KUKA KRL program: MyProgram_263().src

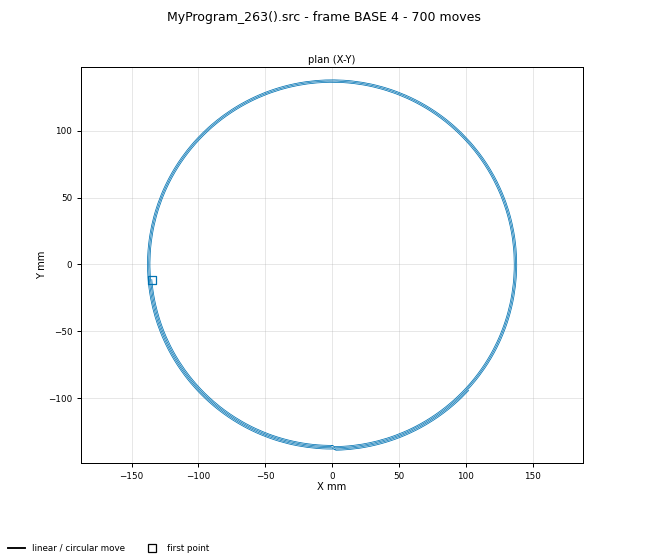
[picture p0: tool path of MyProgram_263().src in frame BASE 4, 700 of 700 moves have a stored position in this frame; points joined in program order, loops and branches not executed]
&ACCESS RVP
&REL 1
&PARAM TEMPLATE = C:\KRC\Roboter\Template\vorgabe
&PARAM EDITMASK = *
DEF MyProgram_263()
; ---- Setting reference (Base) ----
$BASE = BASE_DATA[4]

; --------------------------
; ---- Setting tool (TCP) ----
$TOOL = TOOL_DATA[3]
; --------------------------

$VEL.CP = VEL_APROX_PRINT
Startdeposition()
$VEL.CP = VEL_PRINT
LIN {X -134.8458,Y -11.2904,Z 168,A -173.803,B 10.3704,C 0.1903,E1 10.2126,E2 264.7612} C_DIS
LIN {X -134.4588,Y -15.2399,Z 168,A -171.9605,B 10.3704,C 0.1921,E1 10.2132,E2 262.9003} C_DIS
LIN {X -133.9529,Y -19.1689,Z 168,A -170.374,B 10.3703,C 0.1986,E1 10.2138,E2 261.3266} C_DIS
LIN {X -133.392,Y -22.7512,Z 168,A -168.8018,B 10.3703,C 0.2023,E1 10.2145,E2 259.7513} C_DIS
LIN {X -132.6804,Y -26.5871,Z 168,A -167.1161,B 10.3701,C 0.2064,E1 10.2154,E2 258.0628} C_DIS
LIN {X -131.9635,Y -29.9407,Z 168,A -165.7968,B 10.3701,C 0.213,E1 10.2162,E2 256.7611} C_DIS
LIN {X -130.6956,Y -35.0639,Z 168,A -163.3968,B 10.3699,C 0.2162,E1 10.2178,E2 254.3427} C_DIS
LIN {X -129.3305,Y -39.8048,Z 168,A -161.2288,B 10.3699,C 0.2205,E1 10.2196,E2 252.1668} C_DIS
LIN {X -127.9504,Y -44.0403,Z 168,A -159.3976,B 10.3697,C 0.2267,E1 10.2212,E2 250.3438} C_DIS
LIN {X -126.827,Y -47.1777,Z 168,A -157.8777,B 10.3697,C 0.2284,E1 10.2226,E2 248.8116} C_DIS
LIN {X -125.4357,Y -50.7607,Z 168,A -156.287,B 10.3696,C 0.2335,E1 10.2243,E2 247.2266} C_DIS
LIN {X -123.8895,Y -54.4311,Z 168,A -154.6014,B 10.3695,C 0.238,E1 10.2261,E2 245.5425} C_DIS
LIN {X -120.8002,Y -60.9773,Z 168,A -151.5048,B 10.3693,C 0.2453,E1 10.2299,E2 242.4441} C_DIS
LIN {X -118.8985,Y -64.61,Z 168,A -149.6278,B 10.3693,C 0.247,E1 10.2324,E2 240.551} C_DIS
LIN {X -116.7353,Y -68.4408,Z 168,A -147.7469,B 10.3692,C 0.2512,E1 10.235,E2 238.6689} C_DIS
LIN {X -114.2872,Y -72.4552,Z 168,A -146.0083,B 10.3689,C 0.261,E1 10.2375,E2 236.9629} C_DIS
LIN {X -109.9875,Y -78.8291,Z 168,A -142.3087,B 10.3689,C 0.26,E1 10.2434,E2 233.2102} C_DIS
LIN {X -106.8364,Y -83.0498,Z 168,A -140.2258,B 10.3688,C 0.2679,E1 10.2469,E2 231.1468} C_DIS
LIN {X -104.0676,Y -86.4942,Z 168,A -138.2956,B 10.3687,C 0.2709,E1 10.2503,E2 229.2102} C_DIS
LIN {X -101.2009,Y -89.8315,Z 168,A -136.4119,B 10.3686,C 0.2744,E1 10.2538,E2 227.3247} C_DIS
LIN {X -98.1852,Y -93.1184,Z 168,A -134.4868,B 10.3686,C 0.2776,E1 10.2575,E2 225.3958} C_DIS
LIN {X -95.0955,Y -96.2718,Z 168,A -132.6344,B 10.3684,C 0.2816,E1 10.2611,E2 223.5463} C_DIS
LIN {X -91.911,Y -99.3166,Z 168,A -130.7339,B 10.3684,C 0.2845,E1 10.265,E2 221.642} C_DIS
LIN {X -88.3478,Y -102.4983,Z 168,A -127.9328,B 10.3686,C 0.2721,E1 10.2711,E2 218.7437} C_DIS
LIN {X -83.5517,Y -106.4442,Z 168,A -126.3106,B 10.368,C 0.2976,E1 10.2744,E2 217.2487} C_DIS
LIN {X -80.2823,Y -108.9314,Z 168,A -124.2688,B 10.368,C 0.2942,E1 10.279,E2 215.1697} C_DIS
LIN {X -76.5904,Y -111.5579,Z 168,A -122.3677,B 10.368,C 0.2976,E1 10.2833,E2 213.271} C_DIS
LIN {X -72.4048,Y -114.3191,Z 168,A -119.5332,B 10.3683,C 0.2858,E1 10.2902,E2 210.3474} C_DIS
LIN {X -67.4204,Y -117.3283,Z 168,A -117.9883,B 10.3676,C 0.3086,E1 10.2937,E2 208.9185} C_DIS
LIN {X -64.2373,Y -119.1003,Z 168,A -116.1108,B 10.3678,C 0.3036,E1 10.2984,E2 206.9992} C_DIS
LIN {X -60.1371,Y -121.2202,Z 168,A -114.2859,B 10.3676,C 0.3087,E1 10.3029,E2 205.1905} C_DIS
LIN {X -56.9432,Y -122.7526,Z 168,A -112.8278,B 10.3676,C 0.3112,E1 10.3065,E2 203.7377} C_DIS
LIN {X -51.2127,Y -125.2535,Z 168,A -110.0453,B 10.3676,C 0.3112,E1 10.3137,E2 200.9383} C_DIS
LIN {X -47.9106,Y -126.5525,Z 168,A -108.6757,B 10.3674,C 0.3154,E1 10.3173,E2 199.5851} C_DIS
LIN {X -44.7471,Y -127.7053,Z 168,A -107.1029,B 10.3674,C 0.3134,E1 10.3214,E2 197.9938} C_DIS
LIN {X -40.4758,Y -129.124,Z 168,A -105.146,B 10.3674,C 0.3138,E1 10.3267,E2 196.0302} C_DIS
LIN {X -36.863,Y -130.2001,Z 168,A -103.6169,B 10.3674,C 0.3164,E1 10.3308,E2 194.5092} C_DIS
LIN {X -33.2529,Y -131.1679,Z 168,A -102.06,B 10.3674,C 0.3179,E1 10.3349,E2 192.9552} C_DIS
LIN {X -29.1522,Y -132.1412,Z 168,A -100.2394,B 10.3674,C 0.3181,E1 10.3399,E2 191.1297} C_DIS
LIN {X -25.4818,Y -132.8965,Z 168,A -98.7005,B 10.3673,C 0.3198,E1 10.3441,E2 189.5963} C_DIS
LIN {X -21.682,Y -133.5704,Z 168,A -96.9644,B 10.3673,C 0.3182,E1 10.3489,E2 187.8469} C_DIS
LIN {X -17.6427,Y -134.1624,Z 168,A -95.3562,B 10.3673,C 0.3213,E1 10.3533,E2 186.2533} C_DIS
LIN {X -14.2701,Y -134.5631,Z 168,A -93.9184,B 10.3673,C 0.3216,E1 10.3573,E2 184.8149} C_DIS
LIN {X -10.5281,Y -134.9091,Z 168,A -92.1828,B 10.3673,C 0.3186,E1 10.3622,E2 183.0606} C_DIS
LIN {X -6.8196,Y -135.1457,Z 168,A -90.7307,B 10.3673,C 0.3213,E1 10.3662,E2 181.6231} C_DIS
LIN {X -2.7689,Y -135.2903,Z 168,A -88.9419,B 10.3673,C 0.3196,E1 10.3712,E2 179.8245} C_DIS
LIN {X 0.9792,Y -135.3136,Z 168,A -88.0702,B 10.3668,C 0.3356,E1 10.3735,E2 179.0416} C_DIS
Enddeposition()
LIN {X 0.9792,Y -135.3136,Z 168,A -88.0702,B 10.3668,C 0.3356,E1 10.3735,E2 179.0416} C_DIS
Startdeposition()
$VEL.CP = VEL_PRINT
LIN {X -1.5086,Y -136.2254,Z 168,A -89.0405,B 10.307,C 0.3424,E1 10.311,E2 180.0553} C_DIS
LIN {X -5.484,Y -136.1213,Z 168,A -90.778,B 10.307,C 0.3439,E1 10.3061,E2 181.8016} C_DIS
LIN {X -8.5527,Y -135.963,Z 168,A -92.0736,B 10.307,C 0.3439,E1 10.3025,E2 183.0982} C_DIS
LIN {X -13.1963,Y -135.591,Z 168,A -94.0386,B 10.307,C 0.3438,E1 10.297,E2 185.0647} C_DIS
LIN {X -17.8817,Y -135.0529,Z 168,A -95.9859,B 10.307,C 0.3425,E1 10.2917,E2 187.0081} C_DIS
LIN {X -21.6319,Y -134.5054,Z 168,A -97.5637,B 10.307,C 0.3417,E1 10.2873,E2 188.5845} C_DIS
LIN {X -25.7616,Y -133.7736,Z 168,A -99.3345,B 10.307,C 0.3411,E1 10.2824,E2 190.3565} C_DIS
LIN {X -29.123,Y -133.0826,Z 168,A -100.768,B 10.307,C 0.3402,E1 10.2785,E2 191.7892} C_DIS
LIN {X -32.3071,Y -132.3457,Z 168,A -102.1967,B 10.307,C 0.3406,E1 10.2746,E2 193.225} C_DIS
LIN {X -35.8968,Y -131.4194,Z 168,A -103.7296,B 10.307,C 0.3391,E1 10.2705,E2 194.7551} C_DIS
LIN {X -39.0103,Y -130.5287,Z 168,A -105.0997,B 10.307,C 0.3383,E1 10.2668,E2 196.1263} C_DIS
LIN {X -42.2484,Y -129.5172,Z 168,A -106.5325,B 10.3071,C 0.3374,E1 10.263,E2 197.5601} C_DIS
LIN {X -45.4156,Y -128.4409,Z 168,A -107.9472,B 10.3071,C 0.3364,E1 10.2593,E2 198.976} C_DIS
LIN {X -48.573,Y -127.2804,Z 168,A -109.3701,B 10.3071,C 0.3352,E1 10.2555,E2 200.4} C_DIS
LIN {X -51.7172,Y -126.0356,Z 168,A -110.8009,B 10.3072,C 0.334,E1 10.2518,E2 201.832} C_DIS
LIN {X -54.8451,Y -124.7063,Z 168,A -112.2392,B 10.3072,C 0.3327,E1 10.2481,E2 203.2715} C_DIS
LIN {X -57.4972,Y -123.5035,Z 168,A -113.4678,B 10.3073,C 0.3314,E1 10.245,E2 204.5005} C_DIS
LIN {X -60.8012,Y -121.9117,Z 168,A -115.0386,B 10.3073,C 0.3302,E1 10.2411,E2 206.0748} C_DIS
LIN {X -64.8576,Y -119.8045,Z 168,A -117.0288,B 10.3073,C 0.3292,E1 10.2361,E2 208.0734} C_DIS
LIN {X -68.6292,Y -117.6847,Z 168,A -118.91,B 10.3074,C 0.3281,E1 10.2316,E2 209.9621} C_DIS
LIN {X -72.3466,Y -115.4366,Z 168,A -120.7015,B 10.3075,C 0.3247,E1 10.2273,E2 211.749} C_DIS
LIN {X -75.9181,Y -113.1194,Z 168,A -122.533,B 10.3075,C 0.3229,E1 10.223,E2 213.5853} C_DIS
LIN {X -79.5937,Y -110.5644,Z 168,A -124.4566,B 10.3076,C 0.3207,E1 10.2186,E2 215.5136} C_DIS
LIN {X -83.0341,Y -108.0042,Z 168,A -126.2509,B 10.3077,C 0.3175,E1 10.2146,E2 217.3063} C_DIS
LIN {X -86.5489,Y -105.209,Z 168,A -128.1457,B 10.3078,C 0.3143,E1 10.2105,E2 219.2015} C_DIS
LIN {X -89.9021,Y -102.3584,Z 168,A -130.0271,B 10.3079,C 0.3116,E1 10.2065,E2 221.086} C_DIS
LIN {X -93.1649,Y -99.3979,Z 168,A -131.8853,B 10.308,C 0.3081,E1 10.2027,E2 222.9442} C_DIS
LIN {X -96.3318,Y -96.3318,Z 168,A -133.7845,B 10.3081,C 0.3054,E1 10.1989,E2 224.8484} C_DIS
LIN {X -99.3979,Y -93.1649,Z 168,A -135.6301,B 10.3082,C 0.3015,E1 10.1954,E2 226.6922} C_DIS
LIN {X -102.3584,Y -89.9021,Z 168,A -137.5391,B 10.3082,C 0.2987,E1 10.1918,E2 228.6074} C_DIS
LIN {X -105.209,Y -86.5489,Z 168,A -139.4098,B 10.3084,C 0.295,E1 10.1885,E2 230.4796} C_DIS
LIN {X -107.9455,Y -83.1108,Z 168,A -141.2413,B 10.3085,C 0.2906,E1 10.1853,E2 232.3082} C_DIS
LIN {X -110.5644,Y -79.5937,Z 168,A -143.1423,B 10.3086,C 0.2875,E1 10.1822,E2 234.2152} C_DIS
LIN {X -113.0624,Y -76.0036,Z 168,A -145.0023,B 10.3087,C 0.2835,E1 10.1792,E2 236.0767} C_DIS
LIN {X -115.3278,Y -72.519,Z 168,A -146.7386,B 10.3088,C 0.2791,E1 10.1766,E2 237.8106} C_DIS
LIN {X -117.6847,Y -68.6292,Z 168,A -148.6686,B 10.309,C 0.2747,E1 10.1739,E2 239.7415} C_DIS
LIN {X -119.8045,Y -64.8576,Z 168,A -150.5546,B 10.309,C 0.2715,E1 10.1713,E2 241.6345} C_DIS
LIN {X -121.5696,Y -61.4807,Z 168,A -152.0939,B 10.3092,C 0.2661,E1 10.1694,E2 243.1649} C_DIS
LIN {X -123.2926,Y -57.9533,Z 168,A -153.7231,B 10.3092,C 0.2614,E1 10.1674,E2 244.7903} C_DIS
LIN {X -124.7063,Y -54.8451,Z 168,A -155.1768,B 10.3094,C 0.258,E1 10.1657,E2 246.2451} C_DIS
LIN {X -125.8387,Y -52.1888,Z 168,A -156.4508,B 10.3094,C 0.2559,E1 10.1644,E2 247.5255} C_DIS
LIN {X -127.2804,Y -48.573,Z 168,A -158.0638,B 10.3096,C 0.2511,E1 10.1627,E2 249.1343} C_DIS
LIN {X -128.4409,Y -45.4156,Z 168,A -159.496,B 10.3096,C 0.2476,E1 10.1614,E2 250.5676} C_DIS
LIN {X -129.3486,Y -42.7549,Z 168,A -160.7421,B 10.3096,C 0.2455,E1 10.1602,E2 251.8205} C_DIS
LIN {X -130.5099,Y -39.0744,Z 168,A -162.3371,B 10.3098,C 0.2405,E1 10.1589,E2 253.4107} C_DIS
LIN {X -131.2891,Y -36.3625,Z 168,A -163.5799,B 10.3098,C 0.2382,E1 10.158,E2 254.6594} C_DIS
LIN {X -132.2465,Y -32.7185,Z 168,A -165.1434,B 10.31,C 0.2334,E1 10.1569,E2 256.219} C_DIS
LIN {X -132.8521,Y -30.155,Z 168,A -166.2801,B 10.31,C 0.2308,E1 10.1562,E2 257.3582} C_DIS
LIN {X -133.6569,Y -26.372,Z 168,A -167.9128,B 10.3101,C 0.2263,E1 10.1553,E2 258.9903} C_DIS
LIN {X -134.2422,Y -23.2094,Z 168,A -169.2825,B 10.3101,C 0.2228,E1 10.1546,E2 260.3609} C_DIS
LIN {X -134.9314,Y -18.7824,Z 168,A -171.183,B 10.3103,C 0.2176,E1 10.1538,E2 262.2616} C_DIS
LIN {X -135.2978,Y -15.9235,Z 168,A -172.4765,B 10.3103,C 0.2157,E1 10.1534,E2 263.5639} C_DIS
LIN {X -135.7291,Y -11.6921,Z 168,A -174.2763,B 10.3104,C 0.2107,E1 10.1529,E2 265.3634} C_DIS
LIN {X -135.9751,Y -8.3552,Z 168,A -175.6814,B 10.3105,C 0.2065,E1 10.1526,E2 266.7668} C_DIS
LIN {X -136.1579,Y -4.5455,Z 168,A -177.2807,B 10.3106,C 0.2018,E1 10.1524,E2 268.364} C_DIS
LIN {X -136.2254,Y -1.5086,Z 168,A -178.5008,B 10.3107,C 0.197,E1 10.1524,E2 269.5758} C_DIS
LIN {X -136.2254,Y 1.5086,Z 168,A 179.976,B 10.3107,C 0.198,E1 10.1524,E2 271.1288} C_DIS
LIN {X -136.1281,Y 5.3099,Z 168,A 178.467,B 10.3108,C 0.1917,E1 10.1525,E2 272.6252} C_DIS
LIN {X -135.963,Y 8.5527,Z 168,A 177.0578,B 10.3108,C 0.1885,E1 10.1528,E2 274.0382} C_DIS
LIN {X -135.6827,Y 12.2412,Z 168,A 175.5398,B 10.311,C 0.1832,E1 10.1531,E2 275.5501} C_DIS
LIN {X -135.1791,Y 16.9188,Z 168,A 173.5284,B 10.311,C 0.1781,E1 10.1538,E2 277.5634} C_DIS
LIN {X -134.7492,Y 20.0574,Z 168,A 172.1744,B 10.3111,C 0.1746,E1 10.1543,E2 278.9187} C_DIS
LIN {X -134.2842,Y 22.9573,Z 168,A 170.9468,B 10.3111,C 0.1709,E1 10.1548,E2 280.144} C_DIS
LIN {X -133.7736,Y 25.7616,Z 168,A 169.6915,B 10.3112,C 0.1685,E1 10.1555,E2 281.4049} C_DIS
LIN {X -133.0265,Y 29.383,Z 168,A 168.1143,B 10.3112,C 0.1644,E1 10.1564,E2 282.9831} C_DIS
LIN {X -132.2465,Y 32.7185,Z 168,A 166.6563,B 10.3113,C 0.1607,E1 10.1574,E2 284.4417} C_DIS
LIN {X -131.4194,Y 35.8968,Z 168,A 165.2535,B 10.3113,C 0.1571,E1 10.1584,E2 285.8456} C_DIS
LIN {X -130.5999,Y 38.7669,Z 168,A 163.9581,B 10.3114,C 0.1543,E1 10.1594,E2 287.1446} C_DIS
LIN {X -129.5172,Y 42.2484,Z 168,A 162.4211,B 10.3114,C 0.1501,E1 10.1607,E2 288.6803} C_DIS
LIN {X -128.4409,Y 45.4156,Z 168,A 160.9926,B 10.3115,C 0.1466,E1 10.162,E2 290.11} C_DIS
LIN {X -127.2804,Y 48.573,Z 168,A 159.5563,B 10.3115,C 0.1431,E1 10.1634,E2 291.5473} C_DIS
LIN {X -126.231,Y 51.2325,Z 168,A 158.2884,B 10.3116,C 0.141,E1 10.1647,E2 292.8217} C_DIS
LIN {X -124.7063,Y 54.8451,Z 168,A 156.6623,B 10.3116,C 0.1361,E1 10.1665,E2 294.4434} C_DIS
LIN {X -123.2926,Y 57.9533,Z 168,A 155.2053,B 10.3117,C 0.1327,E1 10.1682,E2 295.9012} C_DIS
LIN {X -121.7947,Y 61.0385,Z 168,A 153.7422,B 10.3117,C 0.1293,E1 10.17,E2 297.3654} C_DIS
LIN {X -119.6923,Y 65.0634,Z 168,A 151.6975,B 10.3118,C 0.1268,E1 10.1727,E2 299.4242} C_DIS
LIN {X -117.4147,Y 69.0887,Z 168,A 149.7862,B 10.3118,C 0.1212,E1 10.1754,E2 301.3293} C_DIS
LIN {X -115.1511,Y 72.799,Z 168,A 147.9336,B 10.3119,C 0.1171,E1 10.1781,E2 303.1829} C_DIS
LIN {X -112.9091,Y 76.2299,Z 168,A 146.1338,B 10.3119,C 0.1143,E1 10.1809,E2 304.99} C_DIS
LIN {X -110.3661,Y 79.8673,Z 168,A 144.268,B 10.312,C 0.1097,E1 10.1839,E2 306.8538} C_DIS
LIN {X -107.7597,Y 83.3506,Z 168,A 142.3971,B 10.312,C 0.1062,E1 10.1871,E2 308.7276} C_DIS
LIN {X -104.9925,Y 86.8103,Z 168,A 140.5192,B 10.312,C 0.1022,E1 10.1904,E2 310.6053} C_DIS
LIN {X -102,Y 90.3075,Z 168,A 138.6132,B 10.3121,C 0.0973,E1 10.1939,E2 312.5057} C_DIS
LIN {X -99.1443,Y 93.4337,Z 168,A 136.7665,B 10.3121,C 0.0947,E1 10.1974,E2 314.3585} C_DIS
LIN {X -96.0906,Y 96.5715,Z 168,A 134.8988,B 10.3121,C 0.0913,E1 10.2011,E2 316.2274} C_DIS
LIN {X -92.7686,Y 99.7669,Z 168,A 132.9897,B 10.3122,C 0.0867,E1 10.2049,E2 318.131} C_DIS
LIN {X -89.6462,Y 102.5818,Z 168,A 131.1553,B 10.3122,C 0.0845,E1 10.2088,E2 319.9716} C_DIS
LIN {X -86.2862,Y 105.4236,Z 168,A 129.2873,B 10.3122,C 0.0814,E1 10.2128,E2 321.8399} C_DIS
LIN {X -82.8419,Y 108.1512,Z 168,A 127.4254,B 10.3122,C 0.0782,E1 10.2169,E2 323.7017} C_DIS
LIN {X -79.2075,Y 110.8405,Z 168,A 125.5335,B 10.3123,C 0.0747,E1 10.2211,E2 325.5905} C_DIS
LIN {X -75.5574,Y 113.3602,Z 168,A 123.6651,B 10.3123,C 0.0716,E1 10.2254,E2 327.4576} C_DIS
LIN {X -71.8927,Y 115.719,Z 168,A 121.8187,B 10.3123,C 0.069,E1 10.2298,E2 329.304} C_DIS
LIN {X -68.3398,Y 117.8522,Z 168,A 120.025,B 10.3123,C 0.0673,E1 10.2341,E2 331.1022} C_DIS
LIN {X -64.5644,Y 119.9621,Z 168,A 118.1946,B 10.3123,C 0.0649,E1 10.2386,E2 332.9323} C_DIS
LIN {X -61.0385,Y 121.7947,Z 168,A 116.5987,B 10.3123,C 0.0611,E1 10.2425,E2 334.5178} C_DIS
LIN {X -58.2028,Y 123.1734,Z 168,A 115.2506,B 10.3124,C 0.0598,E1 10.2459,E2 335.8673} C_DIS
LIN {X -54.8451,Y 124.7063,Z 168,A 113.7046,B 10.3124,C 0.0578,E1 10.2499,E2 337.4114} C_DIS
LIN {X -51.7172,Y 126.0356,Z 168,A 112.2684,B 10.3124,C 0.0563,E1 10.2536,E2 338.8472} C_DIS
LIN {X -49.0658,Y 127.0889,Z 168,A 111.0159,B 10.3124,C 0.056,E1 10.2568,E2 340.105} C_DIS
LIN {X -45.4156,Y 128.4409,Z 168,A 109.4198,B 10.3124,C 0.0535,E1 10.261,E2 341.6951} C_DIS
LIN {X -42.2484,Y 129.5172,Z 168,A 108.0078,B 10.3124,C 0.0522,E1 10.2648,E2 343.1066} C_DIS
LIN {X -39.0744,Y 130.5099,Z 168,A 106.6046,B 10.3124,C 0.0511,E1 10.2685,E2 344.5093} C_DIS
LIN {X -34.9205,Y 131.6797,Z 168,A 104.7668,B 10.3124,C 0.05,E1 10.2735,E2 346.3485} C_DIS
LIN {X -31.1301,Y 132.6294,Z 168,A 103.1379,B 10.3124,C 0.0486,E1 10.2779,E2 347.9747} C_DIS
LIN {X -27.9565,Y 133.3344,Z 168,A 101.7682,B 10.3124,C 0.0477,E1 10.2816,E2 349.3437} C_DIS
LIN {X -25.1268,Y 133.8949,Z 168,A 100.5629,B 10.3124,C 0.0468,E1 10.2849,E2 350.5472} C_DIS
LIN {X -21.6319,Y 134.5054,Z 168,A 99.0596,B 10.3124,C 0.0463,E1 10.289,E2 352.051} C_DIS
LIN {X -18.4863,Y 134.9737,Z 168,A 97.7216,B 10.3124,C 0.0457,E1 10.2927,E2 353.3883} C_DIS
LIN {X -14.3974,Y 135.4687,Z 168,A 96.0097,B 10.3124,C 0.0446,E1 10.2975,E2 355.0966} C_DIS
LIN {X -11.369,Y 135.7564,Z 168,A 94.698,B 10.3124,C 0.0449,E1 10.3011,E2 356.4115} C_DIS
LIN {X -7.6071,Y 136.0212,Z 168,A 93.1255,B 10.3124,C 0.0442,E1 10.3055,E2 357.9816} C_DIS
LIN {X -4.5455,Y 136.1579,Z 168,A 91.8379,B 10.3124,C 0.044,E1 10.3091,E2 359.2684} C_DIS
LIN {X -1.5086,Y 136.2254,Z 168,A 90.4045,B 10.3124,C 0.0473,E1 10.3132,E2 360.7201} C_DIS
LIN {X 2.3553,Y 136.2113,Z 168,A 88.921,B 10.3124,C 0.0442,E1 10.3173,E2 362.1856} C_DIS
LIN {X 5.484,Y 136.1213,Z 168,A 87.554,B 10.3124,C 0.0454,E1 10.3211,E2 363.5582} C_DIS
LIN {X 8.5527,Y 135.963,Z 168,A 86.2595,B 10.3124,C 0.0456,E1 10.3247,E2 364.8525} C_DIS
LIN {X 12.1752,Y 135.6883,Z 168,A 84.8065,B 10.3124,C 0.0443,E1 10.3287,E2 366.296} C_DIS
LIN {X 16.4187,Y 135.2388,Z 168,A 82.9513,B 10.3124,C 0.0461,E1 10.3339,E2 368.1577} C_DIS
LIN {X 20.0574,Y 134.7492,Z 168,A 81.4538,B 10.3124,C 0.0456,E1 10.338,E2 369.6492} C_DIS
LIN {X 23.2094,Y 134.2422,Z 168,A 80.1117,B 10.3124,C 0.0462,E1 10.3417,E2 370.9909} C_DIS
LIN {X 27.43,Y 133.4416,Z 168,A 78.2657,B 10.3124,C 0.048,E1 10.3468,E2 372.841} C_DIS
LIN {X 31.1301,Y 132.6294,Z 168,A 76.7157,B 10.3124,C 0.048,E1 10.351,E2 374.3855} C_DIS
LIN {X 34.3075,Y 131.8432,Z 168,A 75.3415,B 10.3124,C 0.0489,E1 10.3547,E2 375.7591} C_DIS
LIN {X 37.0344,Y 131.1013,Z 168,A 74.1167,B 10.3124,C 0.0506,E1 10.358,E2 376.9881} C_DIS
LIN {X 40.4736,Y 130.0817,Z 168,A 72.6429,B 10.3124,C 0.051,E1 10.3619,E2 378.4574} C_DIS
LIN {X 43.833,Y 128.9896,Z 168,A 71.1698,B 10.3124,C 0.0521,E1 10.3658,E2 379.9289} C_DIS
LIN {X 46.5015,Y 128.0494,Z 168,A 69.937,B 10.3124,C 0.0542,E1 10.3691,E2 381.1666} C_DIS
LIN {X 50.1469,Y 126.6686,Z 168,A 68.3509,B 10.3124,C 0.0546,E1 10.3732,E2 382.7463} C_DIS
LIN {X 53.2834,Y 125.3815,Z 168,A 66.9312,B 10.3124,C 0.056,E1 10.3769,E2 384.1652} C_DIS
LIN {X 56.0342,Y 124.1744,Z 168,A 65.669,B 10.3124,C 0.0574,E1 10.3801,E2 385.4271} C_DIS
LIN {X 59.499,Y 122.5541,Z 168,A 64.0729,B 10.3124,C 0.0591,E1 10.3841,E2 387.0217} C_DIS
LIN {X 62.5714,Y 121.0143,Z 168,A 62.6354,B 10.3124,C 0.0608,E1 10.3877,E2 388.4583} C_DIS
LIN {X 66.6579,Y 118.8116,Z 168,A 60.6087,B 10.3124,C 0.0652,E1 10.3927,E2 390.4941} C_DIS
LIN {X 70.5797,Y 116.5245,Z 168,A 58.7589,B 10.3124,C 0.0666,E1 10.3971,E2 392.337} C_DIS
LIN {X 74.0991,Y 114.3188,Z 168,A 56.9776,B 10.3124,C 0.07,E1 10.4013,E2 394.1227} C_DIS
LIN {X 77.725,Y 111.8852,Z 168,A 55.1543,B 10.3124,C 0.0727,E1 10.4055,E2 395.9447} C_DIS
LIN {X 81.4151,Y 109.2293,Z 168,A 53.2898,B 10.3124,C 0.0748,E1 10.4097,E2 397.8039} C_DIS
LIN {X 84.7611,Y 106.6537,Z 168,A 51.4984,B 10.3123,C 0.0783,E1 10.4136,E2 399.5975} C_DIS
LIN {X 88.1594,Y 103.8623,Z 168,A 49.6622,B 10.3123,C 0.0814,E1 10.4176,E2 401.4326} C_DIS
LIN {X 91.6193,Y 100.8234,Z 168,A 47.7822,B 10.3123,C 0.0837,E1 10.4215,E2 403.3064} C_DIS
LIN {X 94.6601,Y 97.9742,Z 168,A 45.9996,B 10.3123,C 0.0879,E1 10.4251,E2 405.0932} C_DIS
LIN {X 97.9474,Y 94.6878,Z 168,A 44.1112,B 10.3122,C 0.0903,E1 10.4288,E2 406.9742} C_DIS
LIN {X 100.8234,Y 91.6193,Z 168,A 42.3222,B 10.3122,C 0.0945,E1 10.4322,E2 408.7665} C_DIS
LIN {X 103.8623,Y 88.1594,Z 168,A 40.4452,B 10.3122,C 0.0973,E1 10.4356,E2 410.637} C_DIS
LIN {X 106.6537,Y 84.7611,Z 168,A 38.6167,B 10.3121,C 0.1009,E1 10.4388,E2 412.4638} C_DIS
LIN {X 109.2094,Y 81.4418,Z 168,A 36.837,B 10.3121,C 0.1054,E1 10.4418,E2 414.2466} C_DIS
LIN {X 111.8852,Y 77.725,Z 168,A 34.9729,B 10.3121,C 0.1084,E1 10.4448,E2 416.1042} C_DIS
LIN {X 114.2481,Y 74.208,Z 168,A 33.1886,B 10.312,C 0.1127,E1 10.4476,E2 417.8898} C_DIS
LIN {X 116.5245,Y 70.5797,Z 168,A 31.4056,B 10.312,C 0.1167,E1 10.4502,E2 419.6715} C_DIS
LIN {X 118.7116,Y 66.8357,Z 168,A 29.5967,B 10.3119,C 0.1209,E1 10.4527,E2 421.4799} C_DIS
LIN {X 120.8177,Y 62.9457,Z 168,A 27.814,B 10.3119,C 0.1238,E1 10.455,E2 423.2541} C_DIS
LIN {X 122.5541,Y 59.499,Z 168,A 26.2435,B 10.3119,C 0.1267,E1 10.457,E2 424.8194} C_DIS
LIN {X 123.7639,Y 56.9341,Z 168,A 25.059,B 10.3118,C 0.1296,E1 10.4583,E2 426.0036} C_DIS
LIN {X 125.3815,Y 53.2834,Z 168,A 23.4117,B 10.3118,C 0.1333,E1 10.4602,E2 427.6483} C_DIS
LIN {X 126.6686,Y 50.1469,Z 168,A 22.0061,B 10.3117,C 0.1366,E1 10.4616,E2 429.0524} C_DIS
LIN {X 127.8712,Y 46.9957,Z 168,A 20.6081,B 10.3117,C 0.1399,E1 10.463,E2 430.449} C_DIS
LIN {X 128.849,Y 44.2384,Z 168,A 19.3636,B 10.3116,C 0.1436,E1 10.4642,E2 431.6961} C_DIS
LIN {X 130.024,Y 40.662,Z 168,A 17.8361,B 10.3116,C 0.1466,E1 10.4655,E2 433.2181} C_DIS
LIN {X 131.248,Y 36.5097,Z 168,A 16.0431,B 10.3115,C 0.151,E1 10.4669,E2 435.0091} C_DIS
LIN {X 132.1345,Y 33.1597,Z 168,A 14.5712,B 10.3115,C 0.1555,E1 10.4679,E2 436.484} C_DIS
LIN {X 133.2024,Y 28.5683,Z 168,A 12.6697,B 10.3114,C 0.1591,E1 10.469,E2 438.3773} C_DIS
LIN {X 133.8477,Y 25.3735,Z 168,A 11.2772,B 10.3113,C 0.1635,E1 10.4698,E2 439.7736} C_DIS
LIN {X 134.5054,Y 21.6319,Z 168,A 9.7329,B 10.3113,C 0.1668,E1 10.4705,E2 441.3128} C_DIS
LIN {X 134.9737,Y 18.4863,Z 168,A 8.4168,B 10.3112,C 0.1701,E1 10.471,E2 442.6275} C_DIS
LIN {X 135.4687,Y 14.3974,Z 168,A 6.7193,B 10.3112,C 0.1742,E1 10.4716,E2 444.3222} C_DIS
LIN {X 135.7631,Y 11.2891,Z 168,A 5.4204,B 10.3111,C 0.1777,E1 10.4719,E2 445.6206} C_DIS
LIN {X 136.0212,Y 7.6071,Z 168,A 3.893,B 10.311,C 0.1816,E1 10.4722,E2 447.1466} C_DIS
LIN {X 136.2002,Y 3.0238,Z 168,A 1.995,B 10.311,C 0.1865,E1 10.4724,E2 449.0425} C_DIS
LIN {X 136.2359,Y 0,Z 168,A 0.6704,B 10.3108,C 0.1915,E1 10.4724,E2 450.3751} C_DIS
LIN {X 136.1742,Y -3.9586,Z 168,A -0.9026,B 10.3108,C 0.1941,E1 10.4723,E2 451.9381} C_DIS
LIN {X 136.0212,Y -7.6071,Z 168,A -2.4187,B 10.3107,C 0.1981,E1 10.4721,E2 453.4534} C_DIS
LIN {X 135.8136,Y -10.6913,Z 168,A -3.7023,B 10.3107,C 0.2015,E1 10.4718,E2 454.7364} C_DIS
LIN {X 135.4251,Y -14.8026,Z 168,A -5.4338,B 10.3105,C 0.2064,E1 10.4713,E2 456.4689} C_DIS
LIN {X 134.9737,Y -18.4863,Z 168,A -6.9592,B 10.3105,C 0.21,E1 10.4708,E2 457.9916} C_DIS
LIN {X 134.5054,Y -21.6319,Z 168,A -8.2801,B 10.3104,C 0.2135,E1 10.4702,E2 459.3118} C_DIS
LIN {X 133.7736,Y -25.7616,Z 168,A -10.0555,B 10.3103,C 0.2189,E1 10.4693,E2 461.0905} C_DIS
LIN {X 132.992,Y -29.5427,Z 168,A -11.6252,B 10.3103,C 0.2222,E1 10.4684,E2 462.6552} C_DIS
LIN {X 132.2465,Y -32.7185,Z 168,A -12.9801,B 10.3101,C 0.2257,E1 10.4676,E2 464.0096} C_DIS
LIN {X 131.4194,Y -35.8968,Z 168,A -14.3437,B 10.3101,C 0.2292,E1 10.4666,E2 465.3724} C_DIS
LIN {X 130.6207,Y -38.6959,Z 168,A -15.5647,B 10.31,C 0.2326,E1 10.4656,E2 466.5942} C_DIS
LIN {X 129.5172,Y -42.2484,Z 168,A -17.0977,B 10.31,C 0.2362,E1 10.4643,E2 468.1251} C_DIS
LIN {X 128.449,Y -45.3923,Z 168,A -18.477,B 10.3098,C 0.2397,E1 10.4631,E2 469.5038} C_DIS
LIN {X 127.2804,Y -48.573,Z 168,A -19.8843,B 10.3098,C 0.2432,E1 10.4617,E2 470.9105} C_DIS
LIN {X 126.0356,Y -51.7172,Z 168,A -21.289,B 10.3097,C 0.2467,E1 10.4602,E2 472.3146} C_DIS
LIN {X 124.7063,Y -54.8451,Z 168,A -22.7008,B 10.3096,C 0.2501,E1 10.4587,E2 473.7257} C_DIS
LIN {X 123.2926,Y -57.9533,Z 168,A -24.1192,B 10.3095,C 0.2536,E1 10.457,E2 475.1435} C_DIS
LIN {X 121.7947,Y -61.0385,Z 168,A -25.5441,B 10.3095,C 0.257,E1 10.4552,E2 476.5679} C_DIS
LIN {X 120.4771,Y -63.5945,Z 168,A -26.7247,B 10.3093,C 0.2595,E1 10.4537,E2 477.7461} C_DIS
LIN {X 118.5481,Y -67.1267,Z 168,A -28.5242,B 10.3092,C 0.2666,E1 10.4513,E2 479.5608} C_DIS
LIN {X 116.3511,Y -70.8665,Z 168,A -30.3271,B 10.3091,C 0.2707,E1 10.4487,E2 481.3632} C_DIS
LIN {X 114.0271,Y -74.5484,Z 168,A -32.1017,B 10.309,C 0.2739,E1 10.446,E2 483.1327} C_DIS
LIN {X 111.5783,Y -78.1661,Z 168,A -33.9179,B 10.3089,C 0.2779,E1 10.4431,E2 484.9483} C_DIS
LIN {X 109.0074,Y -81.7131,Z 168,A -35.7279,B 10.3088,C 0.2816,E1 10.4401,E2 486.7562} C_DIS
LIN {X 106.3175,Y -85.1835,Z 168,A -37.5656,B 10.3087,C 0.2857,E1 10.437,E2 488.5947} C_DIS
LIN {X 103.5121,Y -88.5714,Z 168,A -39.4309,B 10.3085,C 0.2904,E1 10.4336,E2 490.464} C_DIS
LIN {X 100.595,Y -91.871,Z 168,A -41.263,B 10.3085,C 0.2941,E1 10.4302,E2 492.2955} C_DIS
LIN {X 97.5706,Y -95.0769,Z 168,A -43.061,B 10.3084,C 0.2968,E1 10.4267,E2 494.0885} C_DIS
LIN {X 94.4434,Y -98.1839,Z 168,A -44.9314,B 10.3082,C 0.3011,E1 10.423,E2 495.9629} C_DIS
LIN {X 91.2184,Y -101.1872,Z 168,A -46.7301,B 10.3082,C 0.3036,E1 10.4193,E2 497.7566} C_DIS
LIN {X 87.9007,Y -104.0822,Z 168,A -48.5634,B 10.3081,C 0.3068,E1 10.4154,E2 499.5895} C_DIS
LIN {X 84.4959,Y -106.8648,Z 168,A -50.3944,B 10.308,C 0.31,E1 10.4114,E2 501.4201} C_DIS
LIN {X 81.0096,Y -109.5312,Z 168,A -52.2584,B 10.3079,C 0.3138,E1 10.4072,E2 503.2881} C_DIS
LIN {X 77.448,Y -112.0779,Z 168,A -54.0825,B 10.3078,C 0.3167,E1 10.4031,E2 505.1118} C_DIS
LIN {X 73.817,Y -114.5019,Z 168,A -55.9019,B 10.3077,C 0.3194,E1 10.3988,E2 506.9308} C_DIS
LIN {X 70.123,Y -116.8007,Z 168,A -57.6801,B 10.3077,C 0.3212,E1 10.3946,E2 508.7042} C_DIS
LIN {X 66.3794,Y -118.9681,Z 168,A -59.4846,B 10.3076,C 0.3236,E1 10.3902,E2 510.5085} C_DIS
LIN {X 62.5714,Y -121.0143,Z 168,A -61.2095,B 10.3076,C 0.3241,E1 10.386,E2 512.2234} C_DIS
LIN {X 59.499,Y -122.5541,Z 168,A -62.6437,B 10.3075,C 0.3258,E1 10.3824,E2 513.6574} C_DIS
LIN {X 56.4018,Y -124.01,Z 168,A -64.072,B 10.3075,C 0.3275,E1 10.3788,E2 515.0855} C_DIS
LIN {X 53.2834,Y -125.3815,Z 168,A -65.4942,B 10.3074,C 0.3291,E1 10.3751,E2 516.5076} C_DIS
LIN {X 50.1469,Y -126.6686,Z 168,A -66.91,B 10.3074,C 0.3306,E1 10.3715,E2 517.9233} C_DIS
LIN {X 47.4563,Y -127.6987,Z 168,A -68.1058,B 10.3074,C 0.3316,E1 10.3683,E2 519.118} C_DIS
LIN {X 44.1379,Y -128.8839,Z 168,A -69.6049,B 10.3072,C 0.3336,E1 10.3644,E2 520.6204} C_DIS
LIN {X 40.662,Y -130.024,Z 168,A -71.1143,B 10.3072,C 0.3345,E1 10.3604,E2 522.1274} C_DIS
LIN {X 37.5066,Y -130.9689,Z 168,A -72.4917,B 10.3072,C 0.3356,E1 10.3567,E2 523.5048} C_DIS
LIN {X 34.3075,Y -131.8432,Z 168,A -73.878,B 10.3072,C 0.3366,E1 10.3529,E2 524.8911} C_DIS
LIN {X 31.1301,Y -132.6294,Z 168,A -75.2473,B 10.3072,C 0.3376,E1 10.3492,E2 526.2604} C_DIS
LIN {X 27.9565,Y -133.3344,Z 168,A -76.6075,B 10.3071,C 0.3384,E1 10.3455,E2 527.6206} C_DIS
LIN {X 24.9848,Y -133.9221,Z 168,A -77.8391,B 10.3071,C 0.3384,E1 10.3421,E2 528.8477} C_DIS
LIN {X 22.2403,Y -134.4039,Z 168,A -79.0651,B 10.3071,C 0.3403,E1 10.3388,E2 530.0813} C_DIS
LIN {X 18.4863,Y -134.9737,Z 168,A -80.6314,B 10.3071,C 0.3405,E1 10.3344,E2 531.6447} C_DIS
LIN {X 15.3553,Y -135.3656,Z 168,A -81.953,B 10.3071,C 0.341,E1 10.3308,E2 532.9665} C_DIS
LIN {X 12.2412,Y -135.6827,Z 168,A -83.2649,B 10.307,C 0.3414,E1 10.3271,E2 534.2785} C_DIS
LIN {X 8.3553,Y -135.9751,Z 168,A -84.9225,B 10.307,C 0.3424,E1 10.3225,E2 535.9393} C_DIS
LIN {X 4.5455,Y -136.1579,Z 168,A -86.4967,B 10.307,C 0.3421,E1 10.3181,E2 537.5106} C_DIS
LIN {X 0.9842,Y -136.2283,Z 168,A -87.7957,B 10.3071,C 0.3378,E1 10.3145,E2 538.7853} C_DIS
Enddeposition()
LIN {X 0.9842,Y -136.2283,Z 168,A -87.7957,B 10.3071,C 0.3378,E1 10.3145,E2 538.7853} C_DIS
Startdeposition()
$VEL.CP = VEL_PRINT
LIN {X 2.1064,Y -137.1296,Z 168,A -86.1079,B 10.2483,C 0.3182,E1 10.2602,E2 536.9933} C_DIS
LIN {X 7.988,Y -136.9135,Z 168,A -84.2794,B 10.2479,C 0.3321,E1 10.265,E2 535.245} C_DIS
LIN {X 13.1398,Y -136.5146,Z 168,A -82.1949,B 10.2479,C 0.333,E1 10.2708,E2 533.1687} C_DIS
LIN {X 17.7304,Y -135.9946,Z 168,A -80.3679,B 10.2478,C 0.3344,E1 10.2758,E2 531.3538} C_DIS
LIN {X 21.1226,Y -135.5091,Z 168,A -78.8838,B 10.2478,C 0.3324,E1 10.28,E2 529.8621} C_DIS
LIN {X 24.2246,Y -134.989,Z 168,A -77.245,B 10.2481,C 0.324,E1 10.2846,E2 528.1807} C_DIS
LIN {X 27.8737,Y -134.284,Z 168,A -75.9212,B 10.248,C 0.3282,E1 10.2881,E2 526.8854} C_DIS
LIN {X 31.6426,Y -133.446,Z 168,A -74.4237,B 10.248,C 0.3297,E1 10.2922,E2 525.4015} C_DIS
LIN {X 35.0485,Y -132.5915,Z 168,A -73.0921,B 10.2479,C 0.3317,E1 10.2957,E2 524.0862} C_DIS
LIN {X 38.2334,Y -131.7085,Z 168,A -71.6627,B 10.2479,C 0.3292,E1 10.2996,E2 522.6496} C_DIS
LIN {X 41.4782,Y -130.7228,Z 168,A -70.1958,B 10.248,C 0.3266,E1 10.3035,E2 521.1752} C_DIS
LIN {X 44.6808,Y -129.663,Z 168,A -68.7955,B 10.248,C 0.3254,E1 10.3072,E2 519.775} C_DIS
LIN {X 48.3099,Y -128.355,Z 168,A -67.1836,B 10.2481,C 0.3235,E1 10.3114,E2 518.1618} C_DIS
LIN {X 51.8456,Y -126.9693,Z 168,A -65.5408,B 10.2482,C 0.3203,E1 10.3157,E2 516.5105} C_DIS
LIN {X 55.5542,Y -125.3903,Z 168,A -63.8889,B 10.2482,C 0.3189,E1 10.32,E2 514.8612} C_DIS
LIN {X 58.5669,Y -124.0124,Z 168,A -62.3319,B 10.2485,C 0.3128,E1 10.324,E2 513.2809} C_DIS
LIN {X 65.9178,Y -120.2674,Z 168,A -59.048,B 10.2485,C 0.3118,E1 10.332,E2 510.0149} C_DIS
LIN {X 70.1489,Y -117.8493,Z 168,A -56.5072,B 10.249,C 0.2961,E1 10.3383,E2 507.4073} C_DIS
LIN {X 74.4911,Y -115.154,Z 168,A -54.9388,B 10.2487,C 0.3065,E1 10.3418,E2 505.9099} C_DIS
LIN {X 78.0964,Y -112.7402,Z 168,A -53.2298,B 10.2487,C 0.3059,E1 10.3457,E2 504.2125} C_DIS
LIN {X 81.5005,Y -110.3047,Z 168,A -51.3973,B 10.2488,C 0.3007,E1 10.3499,E2 502.3675} C_DIS
LIN {X 85.0117,Y -107.6219,Z 168,A -49.5603,B 10.2489,C 0.2974,E1 10.354,E2 500.5299} C_DIS
LIN {X 88.538,Y -104.7401,Z 168,A -47.6594,B 10.249,C 0.2937,E1 10.358,E2 498.6273} C_DIS
LIN {X 92.0973,Y -101.6238,Z 168,A -45.7179,B 10.2491,C 0.2906,E1 10.3621,E2 496.6882} C_DIS
LIN {X 95.4119,Y -98.5184,Z 168,A -43.8481,B 10.2492,C 0.2873,E1 10.3659,E2 494.82} C_DIS
LIN {X 98.6871,Y -95.2377,Z 168,A -42.0582,B 10.2492,C 0.2868,E1 10.3693,E2 493.0469} C_DIS
LIN {X 101.2363,Y -92.524,Z 168,A -40.3577,B 10.2494,C 0.2797,E1 10.3726,E2 491.3262} C_DIS
LIN {X 107.497,Y -85.1692,Z 168,A -36.4648,B 10.2496,C 0.2739,E1 10.3796,E2 487.4475} C_DIS
LIN {X 110.2663,Y -81.5524,Z 168,A -34.4735,B 10.2497,C 0.2671,E1 10.3829,E2 485.4428} C_DIS
LIN {X 112.8748,Y -77.902,Z 168,A -32.625,B 10.2498,C 0.2632,E1 10.3859,E2 483.5956} C_DIS
LIN {X 115.4435,Y -74.0414,Z 168,A -30.7434,B 10.2499,C 0.2597,E1 10.3888,E2 481.719} C_DIS
LIN {X 117.3329,Y -71.0093,Z 168,A -29.2808,B 10.25,C 0.2567,E1 10.3909,E2 480.2585} C_DIS
LIN {X 119.6945,Y -66.9524,Z 168,A -27.3262,B 10.2501,C 0.2518,E1 10.3936,E2 478.3027} C_DIS
LIN {X 121.5357,Y -63.5444,Z 168,A -25.376,B 10.2504,C 0.239,E1 10.3962,E2 476.308} C_DIS
LIN {X 123.475,Y -59.6918,Z 168,A -24.1068,B 10.2502,C 0.2478,E1 10.3977,E2 475.1051} C_DIS
LIN {X 125.9603,Y -54.2477,Z 168,A -21.5998,B 10.2504,C 0.2409,E1 10.4005,E2 472.5945} C_DIS
LIN {X 128.1608,Y -48.8283,Z 168,A -19.13,B 10.2506,C 0.2335,E1 10.4031,E2 470.1188} C_DIS
LIN {X 129.4824,Y -45.2016,Z 168,A -17.5764,B 10.2506,C 0.2305,E1 10.4045,E2 468.5708} C_DIS
LIN {X 130.5104,Y -42.143,Z 168,A -16.2104,B 10.2507,C 0.2262,E1 10.4057,E2 467.2012} C_DIS
LIN {X 131.6098,Y -38.5706,Z 168,A -14.8017,B 10.2507,C 0.2257,E1 10.4068,E2 465.8101} C_DIS
LIN {X 132.6313,Y -34.8993,Z 168,A -13.0737,B 10.2509,C 0.2177,E1 10.4081,E2 464.0632} C_DIS
LIN {X 133.6526,Y -30.7553,Z 168,A -11.329,B 10.2509,C 0.2136,E1 10.4092,E2 462.3214} C_DIS
LIN {X 134.4565,Y -27.0259,Z 168,A -9.7985,B 10.251,C 0.2106,E1 10.4101,E2 460.7973} C_DIS
LIN {X 135.6712,Y -20.0661,Z 168,A -6.8228,B 10.2512,C 0.2014,E1 10.4115,E2 457.8155} C_DIS
LIN {X 136.1791,Y -16.2524,Z 168,A -5.3263,B 10.2512,C 0.1996,E1 10.412,E2 456.3314} C_DIS
LIN {X 136.5791,Y -12.468,Z 168,A -3.7319,B 10.2514,C 0.1948,E1 10.4124,E2 454.7347} C_DIS
LIN {X 136.8424,Y -9.1422,Z 168,A -2.2995,B 10.2514,C 0.1898,E1 10.4127,E2 453.2961} C_DIS
LIN {X 137.1206,Y -2.644,Z 168,A 0.1122,B 10.2514,C 0.1897,E1 10.413,E2 450.9203} C_DIS
LIN {X 137.0545,Y 5.0095,Z 168,A 4.0023,B 10.2519,C 0.1625,E1 10.4128,E2 446.9393} C_DIS
LIN {X 136.7985,Y 9.7536,Z 168,A 5.4393,B 10.2518,C 0.1709,E1 10.4125,E2 445.5701} C_DIS
LIN {X 136.5462,Y 12.8113,Z 168,A 6.9338,B 10.2519,C 0.1617,E1 10.4121,E2 444.0473} C_DIS
LIN {X 135.8839,Y 18.5746,Z 168,A 9.1629,B 10.2519,C 0.1597,E1 10.4113,E2 441.8408} C_DIS
LIN {X 135.3451,Y 22.1526,Z 168,A 10.5792,B 10.2519,C 0.1577,E1 10.4107,E2 440.4351} C_DIS
LIN {X 134.6986,Y 25.7901,Z 168,A 12.0451,B 10.252,C 0.1553,E1 10.41,E2 438.9776} C_DIS
LIN {X 133.9134,Y 29.6059,Z 168,A 13.8042,B 10.2521,C 0.1473,E1 10.409,E2 437.2006} C_DIS
LIN {X 132.9787,Y 33.549,Z 168,A 15.3164,B 10.2521,C 0.1471,E1 10.408,E2 435.7096} C_DIS
LIN {X 132.1692,Y 36.6093,Z 168,A 16.6642,B 10.2522,C 0.1428,E1 10.407,E2 434.3575} C_DIS
LIN {X 131.106,Y 40.2499,Z 168,A 18.1926,B 10.2522,C 0.1398,E1 10.4058,E2 432.8349} C_DIS
LIN {X 130.1171,Y 43.3399,Z 168,A 19.5246,B 10.2522,C 0.1366,E1 10.4046,E2 431.5047} C_DIS
LIN {X 129.1497,Y 46.1446,Z 168,A 21.0982,B 10.2524,C 0.1248,E1 10.4031,E2 429.888} C_DIS
LIN {X 127.9302,Y 49.424,Z 168,A 22.2622,B 10.2524,C 0.1284,E1 10.402,E2 428.7606} C_DIS
LIN {X 126.5985,Y 52.7412,Z 168,A 23.7263,B 10.2524,C 0.1251,E1 10.4004,E2 427.299} C_DIS
LIN {X 125.1485,Y 56.0949,Z 168,A 25.1248,B 10.2524,C 0.1243,E1 10.3989,E2 425.9155} C_DIS
LIN {X 123.2546,Y 60.145,Z 168,A 27.1043,B 10.2525,C 0.1166,E1 10.3965,E2 423.9207} C_DIS
LIN {X 121.5655,Y 63.4877,Z 168,A 28.5956,B 10.2525,C 0.1144,E1 10.3946,E2 422.4375} C_DIS
LIN {X 118.9044,Y 68.3466,Z 168,A 30.9859,B 10.2526,C 0.1067,E1 10.3913,E2 420.0363} C_DIS
LIN {X 116.6132,Y 72.1857,Z 168,A 32.8382,B 10.2526,C 0.1025,E1 10.3886,E2 418.1848} C_DIS
LIN {X 114.1333,Y 76.0456,Z 168,A 34.6862,B 10.2527,C 0.0995,E1 10.3858,E2 416.3443} C_DIS
LIN {X 111.6191,Y 79.6901,Z 168,A 36.5173,B 10.2527,C 0.0956,E1 10.3829,E2 414.5145} C_DIS
LIN {X 109.4865,Y 82.5956,Z 168,A 38.0992,B 10.2527,C 0.0903,E1 10.3802,E2 412.9223} C_DIS
LIN {X 106.4843,Y 86.4326,Z 168,A 40.0563,B 10.2528,C 0.0876,E1 10.3768,E2 410.9741} C_DIS
LIN {X 103.5602,Y 89.915,Z 168,A 41.7872,B 10.2528,C 0.0876,E1 10.3737,E2 409.2634} C_DIS
LIN {X 99.6259,Y 94.2552,Z 168,A 44.2764,B 10.2528,C 0.0814,E1 10.369,E2 406.7679} C_DIS
LIN {X 96.6006,Y 97.3532,Z 168,A 46.0179,B 10.2528,C 0.0794,E1 10.3656,E2 405.0342} C_DIS
LIN {X 93.7372,Y 100.1138,Z 168,A 47.8019,B 10.2529,C 0.0731,E1 10.3619,E2 403.2344} C_DIS
LIN {X 90.3291,Y 103.1989,Z 168,A 49.5118,B 10.2529,C 0.0746,E1 10.3584,E2 401.5501} C_DIS
LIN {X 87.3872,Y 105.7015,Z 168,A 51.2091,B 10.2529,C 0.0696,E1 10.3548,E2 399.842} C_DIS
LIN {X 84.5235,Y 108.0053,Z 168,A 52.7932,B 10.2529,C 0.0657,E1 10.3513,E2 398.2514} C_DIS
LIN {X 81.0889,Y 110.6071,Z 168,A 54.5672,B 10.2529,C 0.0632,E1 10.3473,E2 396.4803} C_DIS
LIN {X 77.3397,Y 113.2607,Z 168,A 56.4579,B 10.253,C 0.0608,E1 10.343,E2 394.5928} C_DIS
LIN {X 73.611,Y 115.719,Z 168,A 58.3138,B 10.253,C 0.0581,E1 10.3386,E2 392.7378} C_DIS
LIN {X 69.8234,Y 118.0431,Z 168,A 60.2124,B 10.253,C 0.0544,E1 10.3341,E2 390.8338} C_DIS
LIN {X 65.8828,Y 120.2864,Z 168,A 62.2213,B 10.253,C 0.0491,E1 10.3291,E2 388.8105} C_DIS
LIN {X 61.2061,Y 122.7311,Z 168,A 64.1975,B 10.253,C 0.0516,E1 10.3243,E2 386.8625} C_DIS
LIN {X 58.0146,Y 124.2712,Z 168,A 65.6735,B 10.253,C 0.0499,E1 10.3206,E2 385.3871} C_DIS
LIN {X 55.1266,Y 125.5803,Z 168,A 67.0128,B 10.253,C 0.048,E1 10.3172,E2 384.046} C_DIS
LIN {X 52.1123,Y 126.8609,Z 168,A 68.4245,B 10.253,C 0.0456,E1 10.3135,E2 382.6291} C_DIS
LIN {X 48.4459,Y 128.304,Z 168,A 69.9354,B 10.253,C 0.047,E1 10.3096,E2 381.135} C_DIS
LIN {X 45.185,Y 129.4882,Z 168,A 71.4104,B 10.253,C 0.0451,E1 10.3057,E2 379.6568} C_DIS
LIN {X 41.8913,Y 130.5908,Z 168,A 72.8104,B 10.253,C 0.045,E1 10.302,E2 378.2634} C_DIS
LIN {X 38.39,Y 131.6626,Z 168,A 74.3559,B 10.253,C 0.0434,E1 10.2979,E2 376.7161} C_DIS
LIN {X 34.3623,Y 132.7723,Z 168,A 76.1024,B 10.2531,C 0.0421,E1 10.2932,E2 374.9699} C_DIS
LIN {X 30.6823,Y 133.6692,Z 168,A 77.6722,B 10.2531,C 0.0414,E1 10.2889,E2 373.402} C_DIS
LIN {X 27.4158,Y 134.3772,Z 168,A 79.0609,B 10.2531,C 0.0408,E1 10.2851,E2 372.0146} C_DIS
LIN {X 24.4838,Y 134.9426,Z 168,A 80.2591,B 10.2531,C 0.0413,E1 10.2818,E2 370.8228} C_DIS
LIN {X 20.1518,Y 135.6589,Z 168,A 82.2606,B 10.2531,C 0.0368,E1 10.2763,E2 368.8013} C_DIS
LIN {X 16.2714,Y 136.1768,Z 168,A 83.7737,B 10.2531,C 0.039,E1 10.2721,E2 367.3038} C_DIS
LIN {X 13.0428,Y 136.5239,Z 168,A 85.3914,B 10.2531,C 0.0328,E1 10.2675,E2 365.6543} C_DIS
LIN {X 3.4486,Y 137.1028,Z 168,A 89.1942,B 10.2531,C 0.0371,E1 10.257,E2 361.8796} C_DIS
LIN {X -3.3478,Y 137.1056,Z 168,A 92.1907,B 10.2531,C 0.0339,E1 10.2486,E2 358.8652} C_DIS
LIN {X -7.9247,Y 136.9174,Z 168,A 93.9639,B 10.2531,C 0.0373,E1 10.2437,E2 357.1103} C_DIS
LIN {X -11.9822,Y 136.6218,Z 168,A 95.4905,B 10.2531,C 0.0415,E1 10.2395,E2 355.6059} C_DIS
LIN {X -15.5913,Y 136.258,Z 168,A 97.2037,B 10.2531,C 0.0378,E1 10.2347,E2 353.8693} C_DIS
LIN {X -19.4768,Y 135.7554,Z 168,A 98.7963,B 10.2531,C 0.0394,E1 10.2303,E2 352.283} C_DIS
LIN {X -23.6544,Y 135.0911,Z 168,A 100.5896,B 10.2531,C 0.0398,E1 10.2253,E2 350.4876} C_DIS
LIN {X -27.188,Y 134.4235,Z 168,A 102.0393,B 10.2531,C 0.0418,E1 10.2214,E2 349.0453} C_DIS
LIN {X -30.7357,Y 133.657,Z 168,A 103.5813,B 10.2531,C 0.0423,E1 10.2172,E2 347.5011} C_DIS
LIN {X -34.9653,Y 132.6137,Z 168,A 105.4018,B 10.2531,C 0.0437,E1 10.2123,E2 345.6818} C_DIS
LIN {X -38.0928,Y 131.7497,Z 168,A 106.8117,B 10.2531,C 0.0437,E1 10.2085,E2 344.2662} C_DIS
LIN {X -41.2525,Y 130.7949,Z 168,A 109.0849,B 10.2531,C 0.026,E1 10.2022,E2 341.8832} C_DIS
LIN {X -47.7279,Y 128.573,Z 168,A 110.9763,B 10.2531,C 0.0494,E1 10.1975,E2 340.1142} C_DIS
LIN {X -52.7922,Y 126.5771,Z 168,A 113.1945,B 10.2531,C 0.0531,E1 10.1918,E2 337.9047} C_DIS
LIN {X -55.7682,Y 125.2946,Z 168,A 114.5413,B 10.2531,C 0.0549,E1 10.1883,E2 336.5599} C_DIS
LIN {X -58.7458,Y 123.9269,Z 168,A 115.9738,B 10.2531,C 0.0553,E1 10.1847,E2 335.1208} C_DIS
LIN {X -62.2779,Y 122.1893,Z 168,A 117.743,B 10.2531,C 0.055,E1 10.1802,E2 333.3377} C_DIS
LIN {X -65.948,Y 120.2509,Z 168,A 119.4622,B 10.2531,C 0.0578,E1 10.176,E2 331.6218} C_DIS
LIN {X -69.6667,Y 118.1352,Z 168,A 121.3258,B 10.2531,C 0.0589,E1 10.1715,E2 329.7504} C_DIS
LIN {X -73.3147,Y 115.9064,Z 168,A 123.6078,B 10.2531,C 0.0516,E1 10.1659,E2 327.4087} C_DIS
LIN {X -77.3417,Y 113.2593,Z 168,A 125.1851,B 10.253,C 0.0639,E1 10.1624,E2 325.8873} C_DIS
LIN {X -81.6062,Y 110.2265,Z 168,A 127.8068,B 10.253,C 0.0589,E1 10.1564,E2 323.2138} C_DIS
LIN {X -85.2423,Y 107.4388,Z 168,A 129.1268,B 10.253,C 0.0744,E1 10.1537,E2 321.9691} C_DIS
LIN {X -90.8698,Y 102.7229,Z 168,A 131.9561,B 10.2528,C 0.0851,E1 10.1477,E2 319.1722} C_DIS
LIN {X -95.3984,Y 98.5315,Z 168,A 134.7577,B 10.2528,C 0.0859,E1 10.1419,E2 316.346} C_DIS
LIN {X -98.2992,Y 95.6383,Z 168,A 136.7598,B 10.2528,C 0.0838,E1 10.1379,E2 314.31} C_DIS
LIN {X -101.1024,Y 92.6696,Z 168,A 138.64,B 10.2528,C 0.084,E1 10.1343,E2 312.41} C_DIS
LIN {X -103.256,Y 90.2637,Z 168,A 139.7912,B 10.2528,C 0.091,E1 10.1322,E2 311.2847} C_DIS
LIN {X -106.0072,Y 87.0165,Z 168,A 141.5953,B 10.2528,C 0.0945,E1 10.129,E2 309.4793} C_DIS
LIN {X -108.7242,Y 83.5972,Z 168,A 143.477,B 10.2528,C 0.0976,E1 10.1258,E2 307.5925} C_DIS
LIN {X -111.7643,Y 79.487,Z 168,A 145.6268,B 10.2527,C 0.1025,E1 10.1222,E2 305.4432} C_DIS
LIN {X -114.3238,Y 75.7598,Z 168,A 147.5732,B 10.2527,C 0.106,E1 10.1192,E2 303.4918} C_DIS
LIN {X -116.8184,Y 71.8527,Z 168,A 149.4813,B 10.2526,C 0.1114,E1 10.1164,E2 301.5892} C_DIS
LIN {X -118.97,Y 68.2317,Z 168,A 151.3096,B 10.2526,C 0.1146,E1 10.1138,E2 299.7544} C_DIS
LIN {X -121.163,Y 64.2542,Z 168,A 152.9909,B 10.2525,C 0.1237,E1 10.1116,E2 298.1019} C_DIS
LIN {X -122.9764,Y 60.709,Z 168,A 154.714,B 10.2525,C 0.1269,E1 10.1094,E2 296.3732} C_DIS
LIN {X -124.1503,Y 58.2757,Z 168,A 156.0476,B 10.2525,C 0.126,E1 10.1078,E2 295.0156} C_DIS
LIN {X -125.7814,Y 54.6615,Z 168,A 157.6436,B 10.2524,C 0.1316,E1 10.106,E2 293.4289} C_DIS
LIN {X -127.1325,Y 51.4407,Z 168,A 159.3237,B 10.2524,C 0.1314,E1 10.1042,E2 291.723} C_DIS
LIN {X -129.0912,Y 46.3066,Z 168,A 161.9387,B 10.2524,C 0.1316,E1 10.1016,E2 289.0707} C_DIS
LIN {X -130.5366,Y 42.061,Z 168,A 163.4879,B 10.2522,C 0.1431,E1 10.1003,E2 287.564} C_DIS
LIN {X -132.0043,Y 37.1991,Z 168,A 165.4673,B 10.2521,C 0.1518,E1 10.0988,E2 285.6046} C_DIS
LIN {X -132.9107,Y 33.817,Z 168,A 166.8926,B 10.2521,C 0.1566,E1 10.0978,E2 284.1855} C_DIS
LIN {X -133.768,Y 30.2497,Z 168,A 168.5407,B 10.252,C 0.1588,E1 10.0967,E2 282.5247} C_DIS
LIN {X -134.705,Y 25.7571,Z 168,A 170.5066,B 10.2519,C 0.1634,E1 10.0957,E2 280.5549} C_DIS
LIN {X -135.4714,Y 21.3665,Z 168,A 172.415,B 10.2519,C 0.1679,E1 10.0948,E2 278.6427} C_DIS
LIN {X -136.0813,Y 17.0688,Z 168,A 174.3307,B 10.2518,C 0.1713,E1 10.0941,E2 276.7163} C_DIS
LIN {X -136.6042,Y 12.191,Z 168,A 176.2849,B 10.2516,C 0.1791,E1 10.0935,E2 274.776} C_DIS
LIN {X -136.8681,Y 8.7245,Z 168,A 177.7107,B 10.2516,C 0.1838,E1 10.0933,E2 273.355} C_DIS
LIN {X -137.0418,Y 5.3345,Z 168,A 179.1942,B 10.2516,C 0.1867,E1 10.0931,E2 271.8648} C_DIS
LIN {X -137.1407,Y 1.3281,Z 168,A -179.0034,B 10.2515,C 0.1892,E1 10.093,E2 270.0481} C_DIS
LIN {X -137.1044,Y -3.3892,Z 168,A -176.977,B 10.2514,C 0.1938,E1 10.093,E2 268.0167} C_DIS
LIN {X -136.9084,Y -8.0708,Z 168,A -175.0753,B 10.2512,C 0.2006,E1 10.0934,E2 266.1238} C_DIS
LIN {X -136.6352,Y -11.8233,Z 168,A -173.5268,B 10.2512,C 0.2056,E1 10.0937,E2 264.5798} C_DIS
LIN {X -136.2404,Y -15.7385,Z 168,A -171.822,B 10.2511,C 0.2092,E1 10.0942,E2 262.8689} C_DIS
LIN {X -135.7518,Y -19.5021,Z 168,A -170.2422,B 10.251,C 0.2139,E1 10.0948,E2 261.2912} C_DIS
LIN {X -135.121,Y -23.4871,Z 168,A -168.4461,B 10.251,C 0.2166,E1 10.0956,E2 259.4829} C_DIS
LIN {X -134.4274,Y -27.1688,Z 168,A -166.9804,B 10.2508,C 0.223,E1 10.0964,E2 258.031} C_DIS
LIN {X -133.7341,Y -30.3982,Z 168,A -165.5346,B 10.2508,C 0.2256,E1 10.0973,E2 256.5782} C_DIS
LIN {X -132.8568,Y -34.0293,Z 168,A -163.9334,B 10.2507,C 0.2292,E1 10.0984,E2 254.9732} C_DIS
LIN {X -132.1387,Y -36.7185,Z 168,A -162.0264,B 10.2509,C 0.218,E1 10.0999,E2 252.9734} C_DIS
LIN {X -130.4382,Y -42.369,Z 168,A -160.3319,B 10.2504,C 0.2399,E1 10.1013,E2 251.3782} C_DIS
LIN {X -128.7815,Y -47.1657,Z 168,A -158.1498,B 10.2504,C 0.2444,E1 10.1033,E2 249.1901} C_DIS
LIN {X -127.3527,Y -50.8945,Z 168,A -156.438,B 10.2502,C 0.2481,E1 10.105,E2 247.474} C_DIS
LIN {X -126.0224,Y -54.1041,Z 168,A -154.9653,B 10.2502,C 0.2515,E1 10.1066,E2 245.9997} C_DIS
LIN {X -124.7346,Y -57.0124,Z 168,A -153.5692,B 10.2501,C 0.2537,E1 10.1082,E2 244.5961} C_DIS
LIN {X -123.0561,Y -60.5474,Z 168,A -151.9838,B 10.25,C 0.2589,E1 10.1102,E2 243.018} C_DIS
LIN {X -121.5251,Y -63.5645,Z 168,A -150.5836,B 10.2499,C 0.2627,E1 10.1119,E2 241.6205} C_DIS
LIN {X -119.4866,Y -67.3222,Z 168,A -148.6666,B 10.2499,C 0.2646,E1 10.1146,E2 239.6882} C_DIS
LIN {X -117.1822,Y -71.2584,Z 168,A -146.7066,B 10.2497,C 0.2682,E1 10.1174,E2 237.7226} C_DIS
LIN {X -114.7605,Y -75.0965,Z 168,A -144.7679,B 10.2497,C 0.2719,E1 10.1203,E2 235.7795} C_DIS
LIN {X -112.1831,Y -78.8942,Z 168,A -142.9554,B 10.2494,C 0.2785,E1 10.1232,E2 233.9813} C_DIS
LIN {X -109.9932,Y -81.9195,Z 168,A -141.3127,B 10.2494,C 0.2805,E1 10.1259,E2 232.3291} C_DIS
LIN {X -107.286,Y -85.4344,Z 168,A -139.4338,B 10.2493,C 0.2841,E1 10.1291,E2 230.4479} C_DIS
LIN {X -105.0914,Y -88.1199,Z 168,A -137.7967,B 10.2493,C 0.2834,E1 10.1321,E2 228.7876} C_DIS
LIN {X -101.6038,Y -92.1194,Z 168,A -135.7133,B 10.2491,C 0.2908,E1 10.1359,E2 226.7221} C_DIS
LIN {X -98.4624,Y -95.4698,Z 168,A -133.7779,B 10.2491,C 0.2944,E1 10.1397,E2 224.7853} C_DIS
LIN {X -95.2648,Y -98.6608,Z 168,A -131.8635,B 10.2489,C 0.2976,E1 10.1435,E2 222.8682} C_DIS
LIN {X -91.8862,Y -101.8154,Z 168,A -129.9155,B 10.2489,C 0.3009,E1 10.1475,E2 220.9187} C_DIS
LIN {X -88.6496,Y -104.6452,Z 168,A -128.0892,B 10.2487,C 0.3035,E1 10.1514,E2 219.0891} C_DIS
LIN {X -85.0962,Y -107.5551,Z 168,A -126.1416,B 10.2487,C 0.3063,E1 10.1556,E2 217.1384} C_DIS
LIN {X -81.6094,Y -110.2241,Z 168,A -124.3299,B 10.2486,C 0.3098,E1 10.1596,E2 215.3299} C_DIS
LIN {X -77.988,Y -112.8156,Z 168,A -122.4034,B 10.2486,C 0.3113,E1 10.1641,E2 213.3954} C_DIS
LIN {X -74.2201,Y -115.3291,Z 168,A -120.5084,B 10.2484,C 0.3141,E1 10.1685,E2 211.5003} C_DIS
LIN {X -70.3793,Y -117.712,Z 168,A -118.6151,B 10.2484,C 0.3167,E1 10.173,E2 209.6066} C_DIS
LIN {X -66.2849,Y -120.0652,Z 168,A -116.6477,B 10.2483,C 0.3194,E1 10.1778,E2 207.6401} C_DIS
LIN {X -62.5643,Y -122.0435,Z 168,A -114.928,B 10.2482,C 0.3225,E1 10.182,E2 205.9256} C_DIS
LIN {X -59.3868,Y -123.6207,Z 168,A -113.4791,B 10.2481,C 0.3249,E1 10.1857,E2 204.4809} C_DIS
LIN {X -56.2504,Y -125.079,Z 168,A -112.0251,B 10.2481,C 0.3263,E1 10.1894,E2 203.0257} C_DIS
LIN {X -53.0988,Y -126.4491,Z 168,A -110.5857,B 10.2481,C 0.3277,E1 10.1931,E2 201.5858} C_DIS
LIN {X -49.848,Y -127.7662,Z 168,A -109.1501,B 10.2479,C 0.3298,E1 10.1968,E2 200.1538} C_DIS
LIN {X -46.7574,Y -128.9287,Z 168,A -107.6892,B 10.2479,C 0.3293,E1 10.2006,E2 198.6824} C_DIS
LIN {X -43.3963,Y -130.0983,Z 168,A -106.328,B 10.2479,C 0.3332,E1 10.2042,E2 197.3371} C_DIS
LIN {X -40.4046,Y -131.0586,Z 168,A -104.9734,B 10.2479,C 0.3332,E1 10.2078,E2 195.9769} C_DIS
LIN {X -36.1836,Y -132.2881,Z 168,A -102.9875,B 10.2479,C 0.3313,E1 10.2132,E2 193.9717} C_DIS
LIN {X -32.248,Y -133.3001,Z 168,A -101.3678,B 10.2479,C 0.334,E1 10.2176,E2 192.3616} C_DIS
LIN {X -28.9132,Y -134.063,Z 168,A -99.8643,B 10.2479,C 0.3331,E1 10.2217,E2 190.8481} C_DIS
LIN {X -22.1331,Y -135.3484,Z 168,A -97.0099,B 10.2478,C 0.3349,E1 10.2295,E2 187.9968} C_DIS
LIN {X -18.1145,Y -135.9442,Z 168,A -95.3446,B 10.2478,C 0.3361,E1 10.2341,E2 186.3349} C_DIS
LIN {X -12.5733,Y -136.569,Z 168,A -93.1269,B 10.2476,C 0.339,E1 10.2403,E2 184.1308} C_DIS
LIN {X -6.8457,Y -136.9746,Z 168,A -90.5997,B 10.2477,C 0.3363,E1 10.2473,E2 181.5863} C_DIS
LIN {X 0.9735,Y -137.1384,Z 168,A -88.623,B 10.2468,C 0.3652,E1 10.2525,E2 179.7715} C_DIS
Enddeposition()
LIN {X 0.9735,Y -137.1384,Z 168,A -88.6231,B 10.2468,C 0.3652,E1 10.2525,E2 179.7718} C_DIS
Startdeposition()
$VEL.CP = VEL_PRINT
LIN {X 0.3299,Y -138.06,Z 168,A -88.6706,B 10.1841,C 0.3687,E1 10.1898,E2 179.8458} C_DIS
LIN {X -3.9229,Y -138.0039,Z 168,A -89.9509,B 10.1845,C 0.3579,E1 10.1863,E2 181.0655} C_DIS
LIN {X -7.3523,Y -137.8643,Z 168,A -91.3609,B 10.1845,C 0.3576,E1 10.1824,E2 182.4742} C_DIS
LIN {X -11.2944,Y -137.5972,Z 168,A -93.086,B 10.1845,C 0.3593,E1 10.1775,E2 184.2108} C_DIS
LIN {X -18.7052,Y -136.7886,Z 168,A -96.0892,B 10.1845,C 0.3567,E1 10.1692,E2 187.2038} C_DIS
LIN {X -26.0191,Y -135.5854,Z 168,A -99.5445,B 10.1843,C 0.3639,E1 10.1596,E2 190.7081} C_DIS
LIN {X -29.5489,Y -134.8607,Z 168,A -100.6793,B 10.1846,C 0.3553,E1 10.1566,E2 191.7976} C_DIS
LIN {X -32.8039,Y -134.1063,Z 168,A -102.1564,B 10.1846,C 0.3565,E1 10.1526,E2 193.2865} C_DIS
LIN {X -39.8763,Y -132.1761,Z 168,A -105.0333,B 10.1847,C 0.3509,E1 10.1449,E2 196.143} C_DIS
LIN {X -43.7734,Y -130.9361,Z 168,A -106.8582,B 10.1847,C 0.3523,E1 10.14,E2 197.9843} C_DIS
LIN {X -47.27,Y -129.7155,Z 168,A -108.4063,B 10.1847,C 0.3512,E1 10.1359,E2 199.534} C_DIS
LIN {X -50.3323,Y -128.5583,Z 168,A -109.7647,B 10.1847,C 0.3499,E1 10.1324,E2 200.8925} C_DIS
LIN {X -53.4268,Y -127.3026,Z 168,A -111.1578,B 10.1847,C 0.3487,E1 10.1288,E2 202.2866} C_DIS
LIN {X -56.649,Y -125.9019,Z 168,A -112.6397,B 10.1848,C 0.3476,E1 10.125,E2 203.7715} C_DIS
LIN {X -59.7149,Y -124.4768,Z 168,A -114.0246,B 10.1849,C 0.3457,E1 10.1215,E2 205.1541} C_DIS
LIN {X -62.7931,Y -122.9527,Z 168,A -115.4644,B 10.1849,C 0.3443,E1 10.1179,E2 206.5957} C_DIS
LIN {X -65.9389,Y -121.297,Z 168,A -117.0615,B 10.1849,C 0.3449,E1 10.1139,E2 208.2082} C_DIS
LIN {X -69.8501,Y -119.0875,Z 168,A -118.9314,B 10.185,C 0.3425,E1 10.1094,E2 210.0787} C_DIS
LIN {X -73.8256,Y -116.6648,Z 168,A -120.8679,B 10.185,C 0.3398,E1 10.1048,E2 212.0155} C_DIS
LIN {X -77.7059,Y -114.1175,Z 168,A -122.8241,B 10.1852,C 0.3375,E1 10.1002,E2 213.9752} C_DIS
LIN {X -81.4131,Y -111.5031,Z 168,A -124.6949,B 10.1852,C 0.3343,E1 10.096,E2 215.8442} C_DIS
LIN {X -84.8514,Y -108.9092,Z 168,A -126.5255,B 10.1853,C 0.3321,E1 10.0919,E2 217.6797} C_DIS
LIN {X -88.4404,Y -106.0155,Z 168,A -128.4762,B 10.1854,C 0.3295,E1 10.0877,E2 219.6347} C_DIS
LIN {X -92.2251,Y -102.7396,Z 168,A -130.3023,B 10.1857,C 0.3206,E1 10.0839,E2 221.4284} C_DIS
LIN {X -94.5681,Y -100.5872,Z 168,A -131.8902,B 10.1857,C 0.3235,E1 10.0806,E2 223.0496} C_DIS
LIN {X -97.8857,Y -97.3614,Z 168,A -133.6822,B 10.1858,C 0.3171,E1 10.0771,E2 224.8247} C_DIS
LIN {X -100.6553,Y -94.4959,Z 168,A -135.4876,B 10.1858,C 0.3168,E1 10.0736,E2 226.6486} C_DIS
LIN {X -105.7531,Y -88.7533,Z 168,A -138.5936,B 10.1861,C 0.3084,E1 10.0679,E2 229.7431} C_DIS
LIN {X -108.2675,Y -85.6689,Z 168,A -140.1222,B 10.1863,C 0.3024,E1 10.0652,E2 231.2555} C_DIS
LIN {X -110.2403,Y -83.114,Z 168,A -141.8121,B 10.1861,C 0.3063,E1 10.0623,E2 232.9887} C_DIS
LIN {X -113.1341,Y -79.1305,Z 168,A -143.81,B 10.1863,C 0.3006,E1 10.0591,E2 234.9799} C_DIS
LIN {X -115.6861,Y -75.35,Z 168,A -145.733,B 10.1864,C 0.2967,E1 10.0561,E2 236.9055} C_DIS
LIN {X -118.2104,Y -71.3244,Z 168,A -147.6951,B 10.1866,C 0.2917,E1 10.0532,E2 238.8652} C_DIS
LIN {X -120.4645,Y -67.4479,Z 168,A -149.5371,B 10.1867,C 0.2868,E1 10.0507,E2 240.7037} C_DIS
LIN {X -122.3318,Y -63.9943,Z 168,A -151.1483,B 10.1868,C 0.2823,E1 10.0486,E2 242.3114} C_DIS
LIN {X -123.9684,Y -60.7639,Z 168,A -152.6744,B 10.1869,C 0.2789,E1 10.0467,E2 243.8394} C_DIS
LIN {X -125.4177,Y -57.7128,Z 168,A -154.0975,B 10.187,C 0.2756,E1 10.045,E2 245.2641} C_DIS
LIN {X -126.8571,Y -54.4767,Z 168,A -155.5918,B 10.1871,C 0.2722,E1 10.0433,E2 246.7605} C_DIS
LIN {X -128.1914,Y -51.2584,Z 168,A -157.0676,B 10.1871,C 0.2689,E1 10.0417,E2 248.239} C_DIS
LIN {X -129.7044,Y -47.3007,Z 168,A -158.8455,B 10.1873,C 0.2646,E1 10.04,E2 250.018} C_DIS
LIN {X -130.6167,Y -44.7202,Z 168,A -160.0895,B 10.1873,C 0.2635,E1 10.0389,E2 251.2746} C_DIS
LIN {X -132.3555,Y -39.2763,Z 168,A -162.5337,B 10.1875,C 0.2584,E1 10.0368,E2 253.7259} C_DIS
LIN {X -133.4209,Y -35.4856,Z 168,A -164.0127,B 10.1876,C 0.2508,E1 10.0357,E2 255.1842} C_DIS
LIN {X -134.2125,Y -32.3632,Z 168,A -165.4054,B 10.1877,C 0.2481,E1 10.0348,E2 256.5827} C_DIS
LIN {X -134.988,Y -28.9595,Z 168,A -166.8612,B 10.1878,C 0.2442,E1 10.0339,E2 258.0381} C_DIS
LIN {X -135.6046,Y -25.9188,Z 168,A -168.2117,B 10.1878,C 0.2417,E1 10.0332,E2 259.3953} C_DIS
LIN {X -136.2231,Y -22.4442,Z 168,A -169.7247,B 10.1879,C 0.2384,E1 10.0325,E2 260.913} C_DIS
LIN {X -136.8782,Y -18.0217,Z 168,A -171.5532,B 10.1881,C 0.2326,E1 10.0318,E2 262.7365} C_DIS
LIN {X -137.3282,Y -14.203,Z 168,A -173.1683,B 10.1881,C 0.2283,E1 10.0313,E2 264.3525} C_DIS
LIN {X -137.7253,Y -9.611,Z 168,A -175.2203,B 10.1882,C 0.2254,E1 10.0308,E2 266.42} C_DIS
LIN {X -138.0135,Y -3.5786,Z 168,A -177.6642,B 10.1884,C 0.2169,E1 10.0305,E2 268.8537} C_DIS
LIN {X -138.0468,Y 1.9206,Z 168,A -179.7824,B 10.1886,C 0.2072,E1 10.0305,E2 270.9493} C_DIS
LIN {X -137.9381,Y 5.8079,Z 168,A 178.3359,B 10.1886,C 0.2075,E1 10.0307,E2 272.8626} C_DIS
LIN {X -137.6514,Y 10.6212,Z 168,A 175.9518,B 10.1886,C 0.2088,E1 10.0312,E2 275.292} C_DIS
LIN {X -137.2978,Y 14.4848,Z 168,A 174.9475,B 10.1889,C 0.1928,E1 10.0314,E2 276.2197} C_DIS
LIN {X -136.8037,Y 18.5898,Z 168,A 172.8566,B 10.1889,C 0.1948,E1 10.0322,E2 278.3553} C_DIS
LIN {X -136.1701,Y 22.7618,Z 168,A 171.1892,B 10.1889,C 0.1882,E1 10.0329,E2 280.0105} C_DIS
LIN {X -135.4541,Y 26.7058,Z 168,A 169.5431,B 10.1891,C 0.1831,E1 10.0338,E2 281.6527} C_DIS
LIN {X -134.9547,Y 29.114,Z 168,A 168.4416,B 10.1891,C 0.1816,E1 10.0344,E2 282.7631} C_DIS
LIN {X -134.1686,Y 32.5452,Z 168,A 167.0337,B 10.1891,C 0.1765,E1 10.0353,E2 284.1628} C_DIS
LIN {X -133.346,Y 35.7665,Z 168,A 165.559,B 10.1892,C 0.1743,E1 10.0363,E2 285.6477} C_DIS
LIN {X -132.1658,Y 39.9101,Z 168,A 163.7439,B 10.1893,C 0.1698,E1 10.0378,E2 287.4643} C_DIS
LIN {X -130.3011,Y 45.6306,Z 168,A 161.2908,B 10.1894,C 0.162,E1 10.0399,E2 289.9093} C_DIS
LIN {X -127.8406,Y 52.1287,Z 168,A 158.3482,B 10.1895,C 0.1552,E1 10.0429,E2 292.8561} C_DIS
LIN {X -126.4733,Y 55.3643,Z 168,A 156.8474,B 10.1895,C 0.1521,E1 10.0445,E2 294.3607} C_DIS
LIN {X -124.8529,Y 58.9277,Z 168,A 154.4764,B 10.1895,C 0.1618,E1 10.0475,E2 296.8211} C_DIS
LIN {X -122.3662,Y 63.9289,Z 168,A 153.0779,B 10.1898,C 0.1383,E1 10.0491,E2 298.1045} C_DIS
LIN {X -119.9882,Y 68.2913,Z 168,A 150.6848,B 10.1898,C 0.1393,E1 10.0524,E2 300.5363} C_DIS
LIN {X -117.7027,Y 72.1591,Z 168,A 148.7938,B 10.1898,C 0.1351,E1 10.0551,E2 302.4285} C_DIS
LIN {X -115.2129,Y 76.0715,Z 168,A 146.8703,B 10.1898,C 0.1303,E1 10.058,E2 304.3498} C_DIS
LIN {X -112.6503,Y 79.8176,Z 168,A 144.6895,B 10.1898,C 0.1314,E1 10.0616,E2 306.565} C_DIS
LIN {X -110.5697,Y 82.6757,Z 168,A 143.7211,B 10.19,C 0.1184,E1 10.0631,E2 307.4707} C_DIS
LIN {X -108.7971,Y 84.9951,Z 168,A 142.2225,B 10.19,C 0.1211,E1 10.0657,E2 309.0033} C_DIS
LIN {X -105.9612,Y 88.5051,Z 168,A 140.4767,B 10.19,C 0.1143,E1 10.0687,E2 310.7316} C_DIS
LIN {X -103.4396,Y 91.4389,Z 168,A 138.5774,B 10.19,C 0.1164,E1 10.0723,E2 312.6652} C_DIS
LIN {X -100.612,Y 94.5418,Z 168,A 136.1934,B 10.19,C 0.125,E1 10.077,E2 315.1253} C_DIS
LIN {X -96.2366,Y 98.9922,Z 168,A 133.7965,B 10.19,C 0.1159,E1 10.0817,E2 317.4963} C_DIS
LIN {X -92.5419,Y 102.4546,Z 168,A 132.4478,B 10.1902,C 0.097,E1 10.0843,E2 318.751} C_DIS
LIN {X -90.1482,Y 104.5665,Z 168,A 130.3533,B 10.1902,C 0.1095,E1 10.0889,E2 320.9382} C_DIS
LIN {X -86.3058,Y 107.7604,Z 168,A 128.0489,B 10.1902,C 0.1102,E1 10.094,E2 323.2684} C_DIS
LIN {X -81.4687,Y 111.4621,Z 168,A 126.4427,B 10.1903,C 0.0875,E1 10.0974,E2 324.7602} C_DIS
LIN {X -74.9955,Y 115.9162,Z 168,A 122.5838,B 10.1903,C 0.094,E1 10.1065,E2 328.6892} C_DIS
LIN {X -71.5327,Y 118.0845,Z 168,A 121.3733,B 10.1903,C 0.0816,E1 10.1092,E2 329.839} C_DIS
LIN {X -68.3541,Y 119.9524,Z 168,A 119.679,B 10.1903,C 0.0826,E1 10.1133,E2 331.552} C_DIS
LIN {X -64.0758,Y 122.289,Z 168,A 117.3709,B 10.1903,C 0.0855,E1 10.1191,E2 333.8931} C_DIS
LIN {X -60.7562,Y 123.9722,Z 168,A 116.1848,B 10.1904,C 0.0762,E1 10.122,E2 335.0341} C_DIS
LIN {X -57.7799,Y 125.3867,Z 168,A 114.7876,B 10.1904,C 0.0751,E1 10.1255,E2 336.4338} C_DIS
LIN {X -54.4364,Y 126.8745,Z 168,A 113.1879,B 10.1904,C 0.0749,E1 10.1296,E2 338.0422} C_DIS
LIN {X -50.5608,Y 128.4689,Z 168,A 111.6337,B 10.1904,C 0.0691,E1 10.1336,E2 339.5723} C_DIS
LIN {X -46.9876,Y 129.8173,Z 168,A 109.5408,B 10.1904,C 0.0779,E1 10.1392,E2 341.7261} C_DIS
LIN {X -43.3406,Y 131.0802,Z 168,A 108.1748,B 10.1904,C 0.0715,E1 10.1428,E2 343.0621} C_DIS
LIN {X -39.7603,Y 132.2117,Z 168,A 106.7737,B 10.1904,C 0.0669,E1 10.1464,E2 344.4429} C_DIS
LIN {X -36.359,Y 133.188,Z 168,A 105.1413,B 10.1904,C 0.0691,E1 10.1509,E2 346.0944} C_DIS
LIN {X -32.4653,Y 134.1879,Z 168,A 103.565,B 10.1904,C 0.0659,E1 10.1551,E2 347.6581} C_DIS
LIN {X -28.0707,Y 135.1767,Z 168,A 101.8489,B 10.1905,C 0.0614,E1 10.1597,E2 349.3543} C_DIS
LIN {X -24.1057,Y 135.9388,Z 168,A 99.994,B 10.1905,C 0.0642,E1 10.1649,E2 351.2301} C_DIS
LIN {X -19.7802,Y 136.6353,Z 168,A 97.9955,B 10.1905,C 0.0672,E1 10.1705,E2 353.2495} C_DIS
LIN {X -11.5671,Y 137.5741,Z 168,A 94.8888,B 10.1905,C 0.0591,E1 10.179,E2 356.3147} C_DIS
LIN {X -4.9279,Y 137.9724,Z 168,A 92.1507,B 10.1905,C 0.0581,E1 10.1866,E2 359.0488} C_DIS
LIN {X 1.6209,Y 138.0518,Z 168,A 89.3806,B 10.1905,C 0.0591,E1 10.1944,E2 361.8242} C_DIS
LIN {X 8.6225,Y 137.7901,Z 168,A 86.7676,B 10.1905,C 0.0528,E1 10.2016,E2 364.3996} C_DIS
LIN {X 11.2194,Y 137.6035,Z 168,A 84.9456,B 10.1905,C 0.0694,E1 10.2069,E2 366.3123} C_DIS
LIN {X 14.9488,Y 137.2479,Z 168,A 83.7332,B 10.1905,C 0.0622,E1 10.2101,E2 367.4823} C_DIS
LIN {X 22.7412,Y 136.1736,Z 168,A 80.1906,B 10.1905,C 0.0697,E1 10.22,E2 371.0579} C_DIS
LIN {X 26.1821,Y 135.5543,Z 168,A 79.0953,B 10.1905,C 0.0625,E1 10.2229,E2 372.1093} C_DIS
LIN {X 29.3323,Y 134.9075,Z 168,A 77.7256,B 10.1905,C 0.064,E1 10.2266,E2 373.4829} C_DIS
LIN {X 32.8663,Y 134.0912,Z 168,A 75.6568,B 10.1905,C 0.0776,E1 10.2324,E2 375.6204} C_DIS
LIN {X 37.5417,Y 132.8575,Z 168,A 74.139,B 10.1905,C 0.0681,E1 10.2364,E2 377.078} C_DIS
LIN {X 41.8607,Y 131.5601,Z 168,A 72.3951,B 10.1905,C 0.0668,E1 10.241,E2 378.806} C_DIS
LIN {X 45.0724,Y 130.4946,Z 168,A 70.9497,B 10.1905,C 0.069,E1 10.2448,E2 380.2563} C_DIS
LIN {X 48.6289,Y 129.2115,Z 168,A 69.4114,B 10.1905,C 0.0698,E1 10.2488,E2 381.7907} C_DIS
LIN {X 52.0238,Y 127.8829,Z 168,A 67.9195,B 10.1905,C 0.0709,E1 10.2527,E2 383.2799} C_DIS
LIN {X 54.9113,Y 126.6692,Z 168,A 66.5881,B 10.1905,C 0.073,E1 10.2561,E2 384.615} C_DIS
LIN {X 58.7338,Y 124.9455,Z 168,A 64.7317,B 10.1905,C 0.0778,E1 10.2609,E2 386.4859} C_DIS
LIN {X 62.4957,Y 123.1041,Z 168,A 62.7369,B 10.1903,C 0.0859,E1 10.2659,E2 388.5121} C_DIS
LIN {X 66.1657,Y 121.1733,Z 168,A 61.3754,B 10.1903,C 0.0799,E1 10.2692,E2 389.8297} C_DIS
LIN {X 69.7991,Y 119.1174,Z 168,A 59.64,B 10.1903,C 0.0825,E1 10.2734,E2 391.5655} C_DIS
LIN {X 73.4715,Y 116.8883,Z 168,A 57.8421,B 10.1903,C 0.0855,E1 10.2776,E2 393.3656} C_DIS
LIN {X 77.3446,Y 114.362,Z 168,A 55.9711,B 10.1903,C 0.0874,E1 10.282,E2 395.2309} C_DIS
LIN {X 81.168,Y 111.681,Z 168,A 54.1228,B 10.1903,C 0.0885,E1 10.2862,E2 397.0685} C_DIS
LIN {X 84.2957,Y 109.3399,Z 168,A 52.4507,B 10.1903,C 0.0925,E1 10.2899,E2 398.7472} C_DIS
LIN {X 87.4173,Y 106.8601,Z 168,A 50.603,B 10.1903,C 0.1001,E1 10.294,E2 400.6192} C_DIS
LIN {X 89.9302,Y 104.7543,Z 168,A 49.5876,B 10.1903,C 0.0943,E1 10.296,E2 401.5923} C_DIS
LIN {X 92.8324,Y 102.191,Z 168,A 47.8644,B 10.1903,C 0.1002,E1 10.2996,E2 403.3304} C_DIS
LIN {X 96.9919,Y 98.2528,Z 168,A 45.6364,B 10.1903,C 0.1013,E1 10.3041,E2 405.5408} C_DIS
LIN {X 103.2571,Y 91.6454,Z 168,A 41.8775,B 10.1901,C 0.1088,E1 10.3113,E2 409.299} C_DIS
LIN {X 105.7307,Y 88.78,Z 168,A 40.1205,B 10.1901,C 0.1168,E1 10.3145,E2 411.0798} C_DIS
LIN {X 110.1695,Y 83.2078,Z 168,A 37.6679,B 10.1901,C 0.1111,E1 10.3187,E2 413.4711} C_DIS
LIN {X 113.0718,Y 79.22,Z 168,A 35.2274,B 10.1899,C 0.1256,E1 10.3227,E2 415.9618} C_DIS
LIN {X 115.5969,Y 75.4874,Z 168,A 33.3795,B 10.1899,C 0.1295,E1 10.3256,E2 417.808} C_DIS
LIN {X 117.9653,Y 71.7297,Z 168,A 31.5826,B 10.1899,C 0.1329,E1 10.3282,E2 419.6002} C_DIS
LIN {X 121.1733,Y 66.1657,Z 168,A 29.3137,B 10.1899,C 0.1298,E1 10.3313,E2 421.8213} C_DIS
LIN {X 123.4655,Y 61.7834,Z 168,A 26.792,B 10.1897,C 0.1467,E1 10.3346,E2 424.4029} C_DIS
LIN {X 125.5017,Y 57.5311,Z 168,A 25.0757,B 10.1897,C 0.1459,E1 10.3366,E2 426.0906} C_DIS
LIN {X 127.138,Y 53.8209,Z 168,A 23.3224,B 10.1896,C 0.1521,E1 10.3385,E2 427.854} C_DIS
LIN {X 128.7562,Y 49.8219,Z 168,A 21.351,B 10.1894,C 0.1614,E1 10.3406,E2 429.8493} C_DIS
LIN {X 129.9626,Y 46.5847,Z 168,A 20.2502,B 10.1895,C 0.157,E1 10.3416,E2 430.9096} C_DIS
LIN {X 131.0873,Y 43.3192,Z 168,A 18.8551,B 10.1895,C 0.16,E1 10.3428,E2 432.301} C_DIS
LIN {X 132.0542,Y 40.2747,Z 168,A 17.5193,B 10.1894,C 0.1639,E1 10.3439,E2 433.6392} C_DIS
LIN {X 132.9764,Y 37.1166,Z 168,A 16.1795,B 10.1894,C 0.1671,E1 10.345,E2 434.9769} C_DIS
LIN {X 133.8635,Y 33.7782,Z 168,A 14.779,B 10.1893,C 0.1703,E1 10.3459,E2 436.3744} C_DIS
LIN {X 134.6734,Y 30.3903,Z 168,A 13.0052,B 10.1891,C 0.1827,E1 10.3471,E2 438.1906} C_DIS
LIN {X 135.445,Y 26.7521,Z 168,A 11.8421,B 10.1891,C 0.1775,E1 10.3477,E2 439.3075} C_DIS
LIN {X 135.9538,Y 24.0217,Z 168,A 10.6154,B 10.1891,C 0.1827,E1 10.3483,E2 440.5445} C_DIS
LIN {X 136.6848,Y 19.4344,Z 168,A 8.8516,B 10.1891,C 0.1841,E1 10.349,E2 442.2893} C_DIS
LIN {X 137.2034,Y 15.3623,Z 168,A 6.8919,B 10.1888,C 0.1955,E1 10.3497,E2 444.2829} C_DIS
LIN {X 137.5541,Y 11.8044,Z 168,A 4.8047,B 10.1885,C 0.215,E1 10.3502,E2 446.4468} C_DIS
LIN {X 137.9509,Y 5.4785,Z 168,A 3.1889,B 10.1888,C 0.1971,E1 10.3504,E2 447.9383} C_DIS
LIN {X 138.0573,Y -0.9573,Z 168,A 0.334,B 10.1886,C 0.2096,E1 10.3504,E2 450.8191} C_DIS
LIN {X 137.9587,Y -5.2796,Z 168,A -1.8513,B 10.1883,C 0.2247,E1 10.3503,E2 453.0552} C_DIS
LIN {X 137.714,Y -9.7661,Z 168,A -3.9506,B 10.188,C 0.2361,E1 10.3498,E2 455.1857} C_DIS
LIN {X 137.1639,Y -15.7134,Z 168,A -5.5526,B 10.1883,C 0.2211,E1 10.3494,E2 456.6803} C_DIS
LIN {X 135.9722,Y -23.9189,Z 168,A -9.4128,B 10.1879,C 0.2418,E1 10.3478,E2 460.5971} C_DIS
LIN {X 135.2562,Y -27.6799,Z 168,A -10.2212,B 10.1882,C 0.2266,E1 10.3474,E2 461.3085} C_DIS
LIN {X 134.2632,Y -32.1528,Z 168,A -12.4717,B 10.1879,C 0.2409,E1 10.346,E2 463.6054} C_DIS
LIN {X 132.9943,Y -37.0525,Z 168,A -14.4714,B 10.1879,C 0.2443,E1 10.3445,E2 465.5946} C_DIS
LIN {X 131.9962,Y -40.4644,Z 168,A -16.0378,B 10.1876,C 0.2508,E1 10.3433,E2 467.1741} C_DIS
LIN {X 130.9125,Y -43.8443,Z 168,A -17.4721,B 10.1876,C 0.254,E1 10.342,E2 468.6052} C_DIS
LIN {X 129.6192,Y -47.537,Z 168,A -19.2598,B 10.1874,C 0.2627,E1 10.3403,E2 470.4155} C_DIS
LIN {X 127.9603,Y -51.8318,Z 168,A -20.9363,B 10.1874,C 0.262,E1 10.3386,E2 472.0643} C_DIS
LIN {X 126.4778,Y -55.3539,Z 168,A -22.8267,B 10.1871,C 0.274,E1 10.3365,E2 473.995} C_DIS
LIN {X 124.9829,Y -58.6531,Z 168,A -24.1083,B 10.1871,C 0.2725,E1 10.335,E2 475.2503} C_DIS
LIN {X 123.0082,Y -62.684,Z 168,A -25.8691,B 10.1871,C 0.2749,E1 10.3328,E2 477.0001} C_DIS
LIN {X 121.1198,Y -66.2637,Z 168,A -27.5515,B 10.1869,C 0.2794,E1 10.3306,E2 478.6848} C_DIS
LIN {X 118.9883,Y -70.0189,Z 168,A -29.4724,B 10.1867,C 0.2872,E1 10.3279,E2 480.624} C_DIS
LIN {X 116.5929,Y -73.9395,Z 168,A -31.225,B 10.1867,C 0.2882,E1 10.3253,E2 482.3592} C_DIS
LIN {X 114.0967,Y -77.7366,Z 168,A -33.1163,B 10.1865,C 0.2931,E1 10.3224,E2 484.2532} C_DIS
LIN {X 109.9251,Y -83.5315,Z 168,A -36.0152,B 10.1864,C 0.2986,E1 10.3176,E2 487.1472} C_DIS
LIN {X 107.1716,Y -87.0359,Z 168,A -38.3848,B 10.1859,C 0.3159,E1 10.3133,E2 489.5846} C_DIS
LIN {X 103.785,Y -91.0475,Z 168,A -39.9368,B 10.1862,C 0.3054,E1 10.3106,E2 491.0596} C_DIS
LIN {X 100.1035,Y -95.0806,Z 168,A -42.2593,B 10.186,C 0.3118,E1 10.3062,E2 493.3917} C_DIS
LIN {X 96.7503,Y -98.4898,Z 168,A -44.0753,B 10.186,C 0.3118,E1 10.3026,E2 495.1882} C_DIS
LIN {X 93.8533,Y -101.2547,Z 168,A -46.1759,B 10.1855,C 0.3261,E1 10.2983,E2 497.3463} C_DIS
LIN {X 90.8362,Y -103.9694,Z 168,A -47.1305,B 10.186,C 0.3116,E1 10.2965,E2 498.2097} C_DIS
LIN {X 86.8839,Y -107.2945,Z 168,A -49.6407,B 10.1856,C 0.3248,E1 10.291,E2 500.7689} C_DIS
LIN {X 83.3652,Y -110.0507,Z 168,A -51.81,B 10.1852,C 0.336,E1 10.2861,E2 502.98} C_DIS
LIN {X 80.0408,Y -112.4919,Z 168,A -53.0093,B 10.1855,C 0.3266,E1 10.2835,E2 504.1158} C_DIS
LIN {X 77.0514,Y -114.5605,Z 168,A -54.6796,B 10.1853,C 0.3332,E1 10.2796,E2 505.8082} C_DIS
LIN {X 72.1089,Y -117.7334,Z 168,A -57.1917,B 10.1851,C 0.339,E1 10.2736,E2 508.332} C_DIS
LIN {X 67.1146,Y -120.6506,Z 168,A -59.7978,B 10.1848,C 0.3477,E1 10.2672,E2 510.9665} C_DIS
LIN {X 63.5262,Y -122.5776,Z 168,A -61.0347,B 10.1851,C 0.3393,E1 10.2643,E2 512.1472} C_DIS
LIN {X 58.5843,Y -125.0147,Z 168,A -63.2564,B 10.1851,C 0.3409,E1 10.2587,E2 514.3626} C_DIS
LIN {X 56.0247,Y -126.1812,Z 168,A -64.4543,B 10.185,C 0.3432,E1 10.2557,E2 515.5653} C_DIS
LIN {X 53.1385,Y -127.423,Z 168,A -65.7431,B 10.185,C 0.3445,E1 10.2524,E2 516.8533} C_DIS
LIN {X 50.0657,Y -128.6614,Z 168,A -67.2069,B 10.1848,C 0.3482,E1 10.2485,E2 518.3296} C_DIS
LIN {X 46.589,Y -129.961,Z 168,A -68.6263,B 10.1848,C 0.3471,E1 10.2448,E2 519.7347} C_DIS
LIN {X 43.5414,Y -131.0133,Z 168,A -70.0108,B 10.1848,C 0.3496,E1 10.2412,E2 521.1261} C_DIS
LIN {X 40.1772,Y -132.0841,Z 168,A -71.4605,B 10.1848,C 0.3507,E1 10.2373,E2 522.575} C_DIS
LIN {X 36.9738,Y -133.0163,Z 168,A -72.8234,B 10.1848,C 0.3514,E1 10.2336,E2 523.9362} C_DIS
LIN {X 33.7806,Y -133.8629,Z 168,A -74.1901,B 10.1847,C 0.3525,E1 10.2299,E2 525.3032} C_DIS
LIN {X 30.6339,Y -134.6178,Z 168,A -75.5081,B 10.1847,C 0.353,E1 10.2264,E2 526.6191} C_DIS
LIN {X 22.7228,Y -136.1766,Z 168,A -78.7015,B 10.1847,C 0.3518,E1 10.2177,E2 529.7952} C_DIS
LIN {X 19.6607,Y -136.6524,Z 168,A -80.2084,B 10.1845,C 0.3576,E1 10.2134,E2 531.3311} C_DIS
LIN {X 15.2082,Y -137.22,Z 168,A -81.859,B 10.1846,C 0.3536,E1 10.2089,E2 532.9557} C_DIS
LIN {X 8.9625,Y -137.7692,Z 168,A -84.6462,B 10.1845,C 0.3588,E1 10.2011,E2 535.7681} C_DIS
LIN {X 5.2865,Y -137.9584,Z 168,A -86.2974,B 10.1843,C 0.362,E1 10.1964,E2 537.4359} C_DIS
LIN {X 0.9835,Y -138.0528,Z 168,A -87.4139,B 10.1849,C 0.3471,E1 10.1936,E2 538.4675} C_DIS
Enddeposition()
LIN {X 0.9835,Y -138.0528,Z 168,A -87.4139,B 10.1849,C 0.3471,E1 10.1936,E2 538.4675} C_DIS
Startdeposition()
$VEL.CP = VEL_PRINT
LIN {X 2.9676,Y -138.9435,Z 168,A -86.2611,B 9.9669,C 0.3525,E1 9.9789,E2 537.3694} C_DIS
LIN {X 6.9888,Y -138.7977,Z 168,A -84.6625,B 9.9669,C 0.3535,E1 9.9834,E2 535.7778} C_DIS
LIN {X 13.066,Y -138.3581,Z 168,A -82.0825,B 9.9669,C 0.351,E1 9.9906,E2 533.1876} C_DIS
LIN {X 20.3192,Y -137.4816,Z 168,A -79.1032,B 9.9669,C 0.3503,E1 9.9988,E2 530.2109} C_DIS
LIN {X 23.4407,Y -136.9835,Z 168,A -77.2139,B 9.9675,C 0.3359,E1 10.0043,E2 528.2439} C_DIS
LIN {X 28.8351,Y -135.9499,Z 168,A -75.5059,B 9.9671,C 0.3473,E1 10.0087,E2 526.6075} C_DIS
LIN {X 33.407,Y -134.9007,Z 168,A -73.6411,B 9.9671,C 0.3473,E1 10.0138,E2 524.7505} C_DIS
LIN {X 37.1525,Y -133.9154,Z 168,A -72.0991,B 9.9671,C 0.3472,E1 10.0179,E2 523.2143} C_DIS
LIN {X 40.81,Y -132.8462,Z 168,A -70.5625,B 9.9671,C 0.3465,E1 10.022,E2 521.681} C_DIS
LIN {X 44.2843,Y -131.7293,Z 168,A -68.9688,B 9.9672,C 0.3428,E1 10.0263,E2 520.0746} C_DIS
LIN {X 47.5936,Y -130.5704,Z 168,A -67.653,B 9.9672,C 0.3443,E1 10.0297,E2 518.7746} C_DIS
LIN {X 51.1164,Y -129.2332,Z 168,A -66.0265,B 9.9672,C 0.3408,E1 10.0339,E2 517.1374} C_DIS
LIN {X 54.8134,Y -127.7073,Z 168,A -64.4606,B 9.9672,C 0.3407,E1 10.038,E2 515.5809} C_DIS
LIN {X 58.6017,Y -126.0137,Z 168,A -62.2007,B 9.9678,C 0.3252,E1 10.0439,E2 513.2476} C_DIS
LIN {X 62.8692,Y -123.9395,Z 168,A -60.8194,B 9.9674,C 0.3363,E1 10.0471,E2 511.9399} C_DIS
LIN {X 66.1658,Y -122.2143,Z 168,A -59.1606,B 9.9676,C 0.331,E1 10.0513,E2 510.2636} C_DIS
LIN {X 70.1497,Y -119.9715,Z 168,A -57.3695,B 9.9676,C 0.3304,E1 10.0556,E2 508.4831} C_DIS
LIN {X 75.455,Y -116.7077,Z 168,A -54.7542,B 9.9678,C 0.325,E1 10.0618,E2 505.8593} C_DIS
LIN {X 79.2882,Y -114.1378,Z 168,A -53.0054,B 9.9678,C 0.3254,E1 10.0658,E2 504.1287} C_DIS
LIN {X 83.1568,Y -111.351,Z 168,A -50.8088,B 9.9681,C 0.3162,E1 10.0708,E2 501.9001} C_DIS
LIN {X 86.6559,Y -108.65,Z 168,A -49.124,B 9.9681,C 0.3162,E1 10.0745,E2 500.2315} C_DIS
LIN {X 90.2997,Y -105.6417,Z 168,A -47.3251,B 9.9681,C 0.3159,E1 10.0783,E2 498.4501} C_DIS
LIN {X 94.2501,Y -102.1321,Z 168,A -45.014,B 9.9683,C 0.3082,E1 10.0831,E2 496.1195} C_DIS
LIN {X 97.0045,Y -99.5207,Z 168,A -43.4584,B 9.9684,C 0.3052,E1 10.0862,E2 494.5636} C_DIS
LIN {X 100.2759,Y -96.2231,Z 168,A -41.8003,B 9.9684,C 0.3074,E1 10.0894,E2 492.9369} C_DIS
LIN {X 102.1463,Y -94.2345,Z 168,A -40.3471,B 9.9687,C 0.2967,E1 10.0923,E2 491.4398} C_DIS
Enddeposition()
END
